gfCNCPoint6[7271] = {X 240.3232, Y 30.5783, Z -8.0000, A 0.000, B 0.000, C 0.000 }
gfCNCPoint6[7272] = {X 239.3655, Y 29.5329, Z -8.0000, A 0.000, B 0.000, C 0.000 }
gfCNCPoint6[7273] = {X 238.5491, Y 28.3738, Z -8.0000, A 0.000, B 0.000, C 0.000 }
gfCNCPoint6[7274] = {X 237.8873, Y 27.1200, Z -8.0000, A 0.000, B 0.000, C 0.000 }
gfCNCPoint6[7275] = {X 237.3910, Y 25.7920, Z -8.0000, A 0.000, B 0.000, C 0.000 }
gfCNCPoint6[7276] = {X 236.9772, Y 24.0072, Z -8.0000, A 0.000, B 0.000, C 0.000 }
gfCNCPoint6[7277] = {X 236.7665, Y 22.1872, Z -8.0000, A 0.000, B 0.000, C 0.000 }
gfCNCPoint6[7278] = {X 236.7613, Y 20.3551, Z -8.0000, A 0.000, B 0.000, C 0.000 }
gfCNCPoint6[7279] = {X 236.9619, Y 18.5340, Z -8.0000, A 0.000, B 0.000, C 0.000 }
gfCNCPoint6[7280] = {X 237.3656, Y 16.7468, Z -8.0000, A 0.000, B 0.000, C 0.000 }
gfCNCPoint6[7281] = {X 237.9247, Y 15.2027, Z -8.0000, A 0.000, B 0.000, C 0.000 }
gfCNCPoint6[7282] = {X 238.6960, Y 13.7528, Z -8.0000, A 0.000, B 0.000, C 0.000 }
gfCNCPoint6[7283] = {X 239.6641, Y 12.4263, Z -8.0000, A 0.000, B 0.000, C 0.000 }
gfCNCPoint6[7284] = {X 240.8097, Y 11.2496, Z -8.0000, A 0.000, B 0.000, C 0.000 }
gfCNCPoint6[7285] = {X 242.1099, Y 10.2463, Z -8.0000, A 0.000, B 0.000, C 0.000 }
gfCNCPoint6[7286] = {X 243.5386, Y 9.4365, Z -8.0000, A 0.000, B 0.000, C 0.000 }
gfCNCPoint6[7287] = {X 245.0673, Y 8.8364, Z -8.0000, A 0.000, B 0.000, C 0.000 }
gfCNCPoint6[7288] = {X 246.6653, Y 8.4579, Z -8.0000, A 0.000, B 0.000, C 0.000 }
gfCNCPoint6[7289] = {X 248.7417, Y 8.1890, Z -8.0000, A 0.000, B 0.000, C 0.000 }
gfCNCPoint6[7290] = {X 250.8340, Y 8.1092, Z -8.0000, A 0.000, B 0.000, C 0.000 }
gfCNCPoint6[7291] = {X 266.7614, Y 8.1092, Z -8.0000, A 0.000, B 0.000, C 0.000 }
gfCNCPoint6[7292] = {X 267.6638, Y 8.2176, Z -8.0000, A 0.000, B 0.000, C 0.000 }
gfCNCPoint6[7293] = {X 268.5198, Y 8.5230, Z -8.0000, A 0.000, B 0.000, C 0.000 }
gfCNCPoint6[7294] = {X 269.2870, Y 9.0102, Z -8.0000, A 0.000, B 0.000, C 0.000 }
gfCNCPoint6[7295] = {X 269.9275, Y 9.6550, Z -8.0000, A 0.000, B 0.000, C 0.000 }
gfCNCPoint6[7296] = {X 270.4094, Y 10.4256, Z -8.0000, A 0.000, B 0.000, C 0.000 }
gfCNCPoint6[7297] = {X 270.7088, Y 11.2837, Z -8.0000, A 0.000, B 0.000, C 0.000 }
gfCNCPoint6[7298] = {X 270.8110, Y 12.1867, Z -8.0000, A 0.000, B 0.000, C 0.000 }
gfCNCPoint6[7299] = {X 270.8108, Y 13.0200, Z -8.0000, A 0.000, B 0.000, C 0.000 }
gfCNCPoint6[7300] = {X 270.7023, Y 13.9135, Z -8.0000, A 0.000, B 0.000, C 0.000 }
gfCNCPoint6[7301] = {X 270.4006, Y 14.7615, Z -8.0000, A 0.000, B 0.000, C 0.000 }
gfCNCPoint6[7302] = {X 269.9202, Y 15.5227, Z -8.0000, A 0.000, B 0.000, C 0.000 }
gfCNCPoint6[7303] = {X 269.2847, Y 16.1601, Z -8.0000, A 0.000, B 0.000, C 0.000 }
gfCNCPoint6[7304] = {X 269.2849, Y 28.5938, Z -8.0000, A 0.000, B 0.000, C 0.000 }
gfCNCPoint6[7305] = {X 273.2849, Y 28.5937, Z -8.0000, A 0.000, B 0.000, C 0.000 }
gfCNCPoint6[7306] = {X 269.2049, Y 28.5938, Z -8.0000, A 0.000, B 0.000, C 0.000 }
gfCNCPoint6[7307] = {X 269.2051, Y 41.0652, Z -8.0000, A 0.000, B 0.000, C 0.000 }
gfCNCPoint6[7308] = {X 269.3438, Y 41.1800, Z -8.0000, A 0.000, B 0.000, C 0.000 }
gfCNCPoint6[7309] = {X 269.9292, Y 41.8064, Z -8.0000, A 0.000, B 0.000, C 0.000 }
gfCNCPoint6[7310] = {X 270.3677, Y 42.5431, Z -8.0000, A 0.000, B 0.000, C 0.000 }
gfCNCPoint6[7311] = {X 270.6392, Y 43.3564, Z -8.0000, A 0.000, B 0.000, C 0.000 }
gfCNCPoint6[7312] = {X 270.7310, Y 44.2089, Z -8.0000, A 0.000, B 0.000, C 0.000 }
gfCNCPoint6[7313] = {X 270.7310, Y 45.0000, Z -8.0000, A 0.000, B 0.000, C 0.000 }
gfCNCPoint6[7314] = {X 270.6307, Y 45.8901, Z -8.0000, A 0.000, B 0.000, C 0.000 }
gfCNCPoint6[7315] = {X 270.3349, Y 46.7355, Z -8.0000, A 0.000, B 0.000, C 0.000 }
gfCNCPoint6[7316] = {X 269.8584, Y 47.4940, Z -8.0000, A 0.000, B 0.000, C 0.000 }
gfCNCPoint6[7317] = {X 269.2250, Y 48.1273, Z -8.0000, A 0.000, B 0.000, C 0.000 }
gfCNCPoint6[7318] = {X 268.4666, Y 48.6039, Z -8.0000, A 0.000, B 0.000, C 0.000 }
gfCNCPoint6[7319] = {X 267.6211, Y 48.8997, Z -8.0000, A 0.000, B 0.000, C 0.000 }
gfCNCPoint6[7320] = {X 266.7310, Y 49.0000, Z -8.0000, A 0.000, B 0.000, C 0.000 }
gfCNCPoint6[7321] = {X 260.2876, Y 49.0000, Z -8.0000, A 0.000, B 0.000, C 0.000 }
gfCNCPoint6[7322] = {X 259.3975, Y 48.8997, Z -8.0000, A 0.000, B 0.000, C 0.000 }
gfCNCPoint6[7323] = {X 258.5520, Y 48.6039, Z -8.0000, A 0.000, B 0.000, C 0.000 }
gfCNCPoint6[7324] = {X 257.7936, Y 48.1273, Z -8.0000, A 0.000, B 0.000, C 0.000 }
gfCNCPoint6[7325] = {X 257.1602, Y 47.4939, Z -8.0000, A 0.000, B 0.000, C 0.000 }
gfCNCPoint6[7326] = {X 256.6837, Y 46.7355, Z -8.0000, A 0.000, B 0.000, C 0.000 }
gfCNCPoint6[7327] = {X 256.3878, Y 45.8901, Z -8.0000, A 0.000, B 0.000, C 0.000 }
gfCNCPoint6[7328] = {X 256.2876, Y 45.0000, Z -8.0000, A 0.000, B 0.000, C 0.000 }
gfCNCPoint6[7329] = {X 256.2879, Y 44.1538, Z -8.0000, A 0.000, B 0.000, C 0.000 }
gfCNCPoint6[7330] = {X 256.3986, Y 43.2730, Z -8.0000, A 0.000, B 0.000, C 0.000 }
gfCNCPoint6[7331] = {X 256.7008, Y 42.4382, Z -8.0000, A 0.000, B 0.000, C 0.000 }
gfCNCPoint6[7332] = {X 257.1796, Y 41.6907, Z -8.0000, A 0.000, B 0.000, C 0.000 }
gfCNCPoint6[7333] = {X 257.8115, Y 41.0672, Z -8.0000, A 0.000, B 0.000, C 0.000 }
gfCNCPoint6[7334] = {X 257.8115, Y 34.1538, Z -8.0000, A 0.000, B 0.000, C 0.000 }
gfCNCPoint6[7335] = {X 254.8178, Y 34.1538, Z -8.0000, A 0.000, B 0.000, C 0.000 }
gfCNCPoint6[7336] = {X 254.5738, Y 34.1534, Z -8.0000, A 0.000, B 0.000, C 0.000 }
gfCNCPoint6[7337] = {X 250.1360, Y 42.7967, Z -8.0000, A 0.000, B 0.000, C 0.000 }
gfCNCPoint6[7338] = {X 250.3287, Y 43.4911, Z -8.0000, A 0.000, B 0.000, C 0.000 }
gfCNCPoint6[7339] = {X 250.3936, Y 44.2089, Z -8.0000, A 0.000, B 0.000, C 0.000 }
gfCNCPoint6[7340] = {X 250.3936, Y 45.0000, Z -8.0000, A 0.000, B 0.000, C 0.000 }
gfCNCPoint6[7341] = {X 250.2933, Y 45.8901, Z -8.0000, A 0.000, B 0.000, C 0.000 }
gfCNCPoint6[7342] = {X 249.9974, Y 46.7355, Z -8.0000, A 0.000, B 0.000, C 0.000 }
gfCNCPoint6[7343] = {X 249.5209, Y 47.4940, Z -8.0000, A 0.000, B 0.000, C 0.000 }
gfCNCPoint6[7344] = {X 248.8875, Y 48.1273, Z -8.0000, A 0.000, B 0.000, C 0.000 }
gfCNCPoint6[7345] = {X 248.1291, Y 48.6039, Z -8.0000, A 0.000, B 0.000, C 0.000 }
gfCNCPoint6[7346] = {X 247.2836, Y 48.8997, Z -8.0000, A 0.000, B 0.000, C 0.000 }
gfCNCPoint6[7347] = {X 246.3936, Y 49.0000, Z -8.0000, A 0.000, B 0.000, C 0.000 }
gfCNCPoint6[7348] = {X 239.8075, Y 49.0000, Z -8.0000, A 0.000, B 0.000, C 0.000 }
gfCNCPoint6[7349] = {X 238.9174, Y 48.8997, Z -8.0000, A 0.000, B 0.000, C 0.000 }
gfCNCPoint6[7350] = {X 238.0720, Y 48.6039, Z -8.0000, A 0.000, B 0.000, C 0.000 }
gfCNCPoint6[7351] = {X 237.3135, Y 48.1273, Z -8.0000, A 0.000, B 0.000, C 0.000 }
gfCNCPoint6[7352] = {X 236.6802, Y 47.4940, Z -8.0000, A 0.000, B 0.000, C 0.000 }
gfCNCPoint6[7353] = {X 236.2036, Y 46.7355, Z -8.0000, A 0.000, B 0.000, C 0.000 }
gfCNCPoint6[7354] = {X 235.9078, Y 45.8901, Z -8.0000, A 0.000, B 0.000, C 0.000 }
gfCNCPoint6[7355] = {X 235.8075, Y 45.0000, Z -8.0000, A 0.000, B 0.000, C 0.000 }
gfCNCPoint6[7356] = {X 235.8079, Y 44.1538, Z -8.0000, A 0.000, B 0.000, C 0.000 }
gfCNCPoint6[7357] = {X 235.9027, Y 43.3414, Z -8.0000, A 0.000, B 0.000, C 0.000 }
gfCNCPoint6[7358] = {X 236.1607, Y 42.5654, Z -8.0000, A 0.000, B 0.000, C 0.000 }
gfCNCPoint6[7359] = {X 236.5712, Y 41.8580, Z -8.0000, A 0.000, B 0.000, C 0.000 }
gfCNCPoint6[7360] = {X 237.1169, Y 41.2489, Z -8.0000, A 0.000, B 0.000, C 0.000 }
gfCNCPoint6[7361] = {X 237.7752, Y 40.7635, Z -8.0000, A 0.000, B 0.000, C 0.000 }
gfCNCPoint6[7362] = {X 238.5184, Y 40.4222, Z -8.0000, A 0.000, B 0.000, C 0.000 }
gfCNCPoint6[7363] = {X 242.7041, Y 32.2292, Z -8.0000, A 0.000, B 0.000, C 0.000 }
gfCNCPoint6[7364] = {X 241.5058, Y 31.4666, Z -8.0000, A 0.000, B 0.000, C 0.000 }
gfCNCPoint6[7365] = {X 240.4158, Y 30.5561, Z -8.0000, A 0.000, B 0.000, C 0.000 }
gfCNCPoint6[7366] = {X 239.4521, Y 29.5127, Z -8.0000, A 0.000, B 0.000, C 0.000 }
gfCNCPoint6[7367] = {X 238.6308, Y 28.3539, Z -8.0000, A 0.000, B 0.000, C 0.000 }
gfCNCPoint6[7368] = {X 237.9656, Y 27.0990, Z -8.0000, A 0.000, B 0.000, C 0.000 }
gfCNCPoint6[7369] = {X 237.4676, Y 25.7689, Z -8.0000, A 0.000, B 0.000, C 0.000 }
gfCNCPoint6[7370] = {X 237.0560, Y 23.9929, Z -8.0000, A 0.000, B 0.000, C 0.000 }
gfCNCPoint6[7371] = {X 236.8463, Y 22.1820, Z -8.0000, A 0.000, B 0.000, C 0.000 }
gfCNCPoint6[7372] = {X 236.8412, Y 20.3590, Z -8.0000, A 0.000, B 0.000, C 0.000 }
gfCNCPoint6[7373] = {X 237.0408, Y 18.5469, Z -8.0000, A 0.000, B 0.000, C 0.000 }
gfCNCPoint6[7374] = {X 237.4426, Y 16.7687, Z -8.0000, A 0.000, B 0.000, C 0.000 }
gfCNCPoint6[7375] = {X 237.9978, Y 15.2351, Z -8.0000, A 0.000, B 0.000, C 0.000 }
gfCNCPoint6[7376] = {X 238.7638, Y 13.7952, Z -8.0000, A 0.000, B 0.000, C 0.000 }
gfCNCPoint6[7377] = {X 239.7254, Y 12.4778, Z -8.0000, A 0.000, B 0.000, C 0.000 }
gfCNCPoint6[7378] = {X 240.8631, Y 11.3092, Z -8.0000, A 0.000, B 0.000, C 0.000 }
gfCNCPoint6[7379] = {X 242.1544, Y 10.3128, Z -8.0000, A 0.000, B 0.000, C 0.000 }
gfCNCPoint6[7380] = {X 243.5734, Y 9.5086, Z -8.0000, A 0.000, B 0.000, C 0.000 }
gfCNCPoint6[7381] = {X 245.0916, Y 8.9126, Z -8.0000, A 0.000, B 0.000, C 0.000 }
gfCNCPoint6[7382] = {X 246.6787, Y 8.5367, Z -8.0000, A 0.000, B 0.000, C 0.000 }
gfCNCPoint6[7383] = {X 248.7483, Y 8.2687, Z -8.0000, A 0.000, B 0.000, C 0.000 }
gfCNCPoint6[7384] = {X 250.8336, Y 8.1892, Z -8.0000, A 0.000, B 0.000, C 0.000 }
gfCNCPoint6[7385] = {X 266.7608, Y 8.1892, Z -8.0000, A 0.000, B 0.000, C 0.000 }
gfCNCPoint6[7386] = {X 267.6454, Y 8.2955, Z -8.0000, A 0.000, B 0.000, C 0.000 }
gfCNCPoint6[7387] = {X 268.4847, Y 8.5949, Z -8.0000, A 0.000, B 0.000, C 0.000 }
gfCNCPoint6[7388] = {X 269.2369, Y 9.0725, Z -8.0000, A 0.000, B 0.000, C 0.000 }
gfCNCPoint6[7389] = {X 269.8648, Y 9.7047, Z -8.0000, A 0.000, B 0.000, C 0.000 }
gfCNCPoint6[7390] = {X 270.3372, Y 10.4602, Z -8.0000, A 0.000, B 0.000, C 0.000 }
gfCNCPoint6[7391] = {X 270.6308, Y 11.3015, Z -8.0000, A 0.000, B 0.000, C 0.000 }
gfCNCPoint6[7392] = {X 270.7310, Y 12.1868, Z -8.0000, A 0.000, B 0.000, C 0.000 }
gfCNCPoint6[7393] = {X 270.7308, Y 13.0192, Z -8.0000, A 0.000, B 0.000, C 0.000 }
gfCNCPoint6[7394] = {X 270.6223, Y 13.9045, Z -8.0000, A 0.000, B 0.000, C 0.000 }
gfCNCPoint6[7395] = {X 270.3202, Y 14.7437, Z -8.0000, A 0.000, B 0.000, C 0.000 }
gfCNCPoint6[7396] = {X 269.8397, Y 15.4952, Z -8.0000, A 0.000, B 0.000, C 0.000 }
gfCNCPoint6[7397] = {X 269.2047, Y 16.1215, Z -8.0000, A 0.000, B 0.000, C 0.000 }
gfCNCPoint6[7398] = {X 269.2049, Y 28.5938, Z -8.0000, A 0.000, B 0.000, C 0.000 }
gfCNCPoint6[7399] = {X 273.2849, Y 28.5937, Z -8.0000, A 0.000, B 0.000, C 0.000 }
gfCNCPoint6[7400] = {X 273.2849, Y 28.5937, Z -5.0000, A 0.000, B 0.000, C 0.000 }
gfCNCPoint6[7401] = {X 273.2849, Y 28.5937, Z 11.0000, A 0.000, B 0.000, C 0.000 }
gfCNCPoint6[7402] = {X 277.7442, Y 28.5918, Z 11.0000, A 0.000, B 0.000, C 0.000 }
gfCNCPoint6[7403] = {X 277.7442, Y 28.5918, Z -5.0000, A 0.000, B 0.000, C 0.000 }
gfCNCPoint6[7404] = {X 277.7442, Y 28.5918, Z -8.0000, A 0.000, B 0.000, C 0.000 }
gfCNCPoint6[7405] = {X 281.8242, Y 28.5918, Z -8.0000, A 0.000, B 0.000, C 0.000 }
gfCNCPoint6[7406] = {X 281.8243, Y 16.2734, Z -8.0000, A 0.000, B 0.000, C 0.000 }
gfCNCPoint6[7407] = {X 281.1862, Y 15.6023, Z -8.0000, A 0.000, B 0.000, C 0.000 }
gfCNCPoint6[7408] = {X 280.7057, Y 14.8107, Z -8.0000, A 0.000, B 0.000, C 0.000 }
gfCNCPoint6[7409] = {X 280.4050, Y 13.9349, Z -8.0000, A 0.000, B 0.000, C 0.000 }
gfCNCPoint6[7410] = {X 280.2978, Y 13.0151, Z -8.0000, A 0.000, B 0.000, C 0.000 }
gfCNCPoint6[7411] = {X 280.2977, Y 12.1868, Z -8.0000, A 0.000, B 0.000, C 0.000 }
gfCNCPoint6[7412] = {X 280.4060, Y 11.2255, Z -8.0000, A 0.000, B 0.000, C 0.000 }
gfCNCPoint6[7413] = {X 280.7255, Y 10.3124, Z -8.0000, A 0.000, B 0.000, C 0.000 }
gfCNCPoint6[7414] = {X 281.2402, Y 9.4933, Z -8.0000, A 0.000, B 0.000, C 0.000 }
gfCNCPoint6[7415] = {X 281.9242, Y 8.8093, Z -8.0000, A 0.000, B 0.000, C 0.000 }
gfCNCPoint6[7416] = {X 282.7433, Y 8.2946, Z -8.0000, A 0.000, B 0.000, C 0.000 }
gfCNCPoint6[7417] = {X 283.6564, Y 7.9751, Z -8.0000, A 0.000, B 0.000, C 0.000 }
gfCNCPoint6[7418] = {X 284.6177, Y 7.8668, Z -8.0000, A 0.000, B 0.000, C 0.000 }
gfCNCPoint6[7419] = {X 291.0611, Y 7.8668, Z -8.0000, A 0.000, B 0.000, C 0.000 }
gfCNCPoint6[7420] = {X 292.0224, Y 7.9751, Z -8.0000, A 0.000, B 0.000, C 0.000 }
gfCNCPoint6[7421] = {X 292.9355, Y 8.2946, Z -8.0000, A 0.000, B 0.000, C 0.000 }
gfCNCPoint6[7422] = {X 293.7546, Y 8.8093, Z -8.0000, A 0.000, B 0.000, C 0.000 }
gfCNCPoint6[7423] = {X 294.4386, Y 9.4933, Z -8.0000, A 0.000, B 0.000, C 0.000 }
gfCNCPoint6[7424] = {X 294.9533, Y 10.3124, Z -8.0000, A 0.000, B 0.000, C 0.000 }
gfCNCPoint6[7425] = {X 295.2728, Y 11.2255, Z -8.0000, A 0.000, B 0.000, C 0.000 }
gfCNCPoint6[7426] = {X 295.3811, Y 12.1868, Z -8.0000, A 0.000, B 0.000, C 0.000 }
gfCNCPoint6[7427] = {X 295.3811, Y 12.9782, Z -8.0000, A 0.000, B 0.000, C 0.000 }
gfCNCPoint6[7428] = {X 295.2798, Y 13.9077, Z -8.0000, A 0.000, B 0.000, C 0.000 }
gfCNCPoint6[7429] = {X 294.9809, Y 14.7936, Z -8.0000, A 0.000, B 0.000, C 0.000 }
gfCNCPoint6[7430] = {X 294.4983, Y 15.5945, Z -8.0000, A 0.000, B 0.000, C 0.000 }
gfCNCPoint6[7431] = {X 293.8548, Y 16.2728, Z -8.0000, A 0.000, B 0.000, C 0.000 }
gfCNCPoint6[7432] = {X 293.8557, Y 22.1965, Z -8.0000, A 0.000, B 0.000, C 0.000 }
gfCNCPoint6[7433] = {X 302.7582, Y 22.1965, Z -8.0000, A 0.000, B 0.000, C 0.000 }
gfCNCPoint6[7434] = {X 302.7633, Y 16.2771, Z -8.0000, A 0.000, B 0.000, C 0.000 }
gfCNCPoint6[7435] = {X 302.1236, Y 15.6061, Z -8.0000, A 0.000, B 0.000, C 0.000 }
gfCNCPoint6[7436] = {X 301.6418, Y 14.8140, Z -8.0000, A 0.000, B 0.000, C 0.000 }
gfCNCPoint6[7437] = {X 301.3401, Y 13.9374, Z -8.0000, A 0.000, B 0.000, C 0.000 }
gfCNCPoint6[7438] = {X 301.2324, Y 13.0165, Z -8.0000, A 0.000, B 0.000, C 0.000 }
gfCNCPoint6[7439] = {X 301.2323, Y 12.1868, Z -8.0000, A 0.000, B 0.000, C 0.000 }
gfCNCPoint6[7440] = {X 301.3406, Y 11.2255, Z -8.0000, A 0.000, B 0.000, C 0.000 }
gfCNCPoint6[7441] = {X 301.6601, Y 10.3124, Z -8.0000, A 0.000, B 0.000, C 0.000 }
gfCNCPoint6[7442] = {X 302.1747, Y 9.4933, Z -8.0000, A 0.000, B 0.000, C 0.000 }
gfCNCPoint6[7443] = {X 302.8588, Y 8.8093, Z -8.0000, A 0.000, B 0.000, C 0.000 }
gfCNCPoint6[7444] = {X 303.6779, Y 8.2946, Z -8.0000, A 0.000, B 0.000, C 0.000 }
gfCNCPoint6[7445] = {X 304.5910, Y 7.9751, Z -8.0000, A 0.000, B 0.000, C 0.000 }
gfCNCPoint6[7446] = {X 305.5523, Y 7.8668, Z -8.0000, A 0.000, B 0.000, C 0.000 }
gfCNCPoint6[7447] = {X 311.9957, Y 7.8668, Z -8.0000, A 0.000, B 0.000, C 0.000 }
gfCNCPoint6[7448] = {X 312.9570, Y 7.9751, Z -8.0000, A 0.000, B 0.000, C 0.000 }
gfCNCPoint6[7449] = {X 313.8701, Y 8.2946, Z -8.0000, A 0.000, B 0.000, C 0.000 }
gfCNCPoint6[7450] = {X 314.6892, Y 8.8093, Z -8.0000, A 0.000, B 0.000, C 0.000 }
gfCNCPoint6[7451] = {X 315.3732, Y 9.4933, Z -8.0000, A 0.000, B 0.000, C 0.000 }
gfCNCPoint6[7452] = {X 315.8879, Y 10.3124, Z -8.0000, A 0.000, B 0.000, C 0.000 }
gfCNCPoint6[7453] = {X 316.2074, Y 11.2255, Z -8.0000, A 0.000, B 0.000, C 0.000 }
gfCNCPoint6[7454] = {X 316.3157, Y 12.1868, Z -8.0000, A 0.000, B 0.000, C 0.000 }
gfCNCPoint6[7455] = {X 316.3157, Y 12.9782, Z -8.0000, A 0.000, B 0.000, C 0.000 }
gfCNCPoint6[7456] = {X 316.2145, Y 13.9077, Z -8.0000, A 0.000, B 0.000, C 0.000 }
gfCNCPoint6[7457] = {X 315.9156, Y 14.7937, Z -8.0000, A 0.000, B 0.000, C 0.000 }
gfCNCPoint6[7458] = {X 315.4331, Y 15.5947, Z -8.0000, A 0.000, B 0.000, C 0.000 }
gfCNCPoint6[7459] = {X 314.7895, Y 16.2730, Z -8.0000, A 0.000, B 0.000, C 0.000 }
gfCNCPoint6[7460] = {X 314.7893, Y 40.9136, Z -8.0000, A 0.000, B 0.000, C 0.000 }
gfCNCPoint6[7461] = {X 315.4273, Y 41.5845, Z -8.0000, A 0.000, B 0.000, C 0.000 }
gfCNCPoint6[7462] = {X 315.9077, Y 42.3760, Z -8.0000, A 0.000, B 0.000, C 0.000 }
gfCNCPoint6[7463] = {X 316.2084, Y 43.2517, Z -8.0000, A 0.000, B 0.000, C 0.000 }
gfCNCPoint6[7464] = {X 316.3156, Y 44.1713, Z -8.0000, A 0.000, B 0.000, C 0.000 }
gfCNCPoint6[7465] = {X 316.3157, Y 45.0000, Z -8.0000, A 0.000, B 0.000, C 0.000 }
gfCNCPoint6[7466] = {X 316.2074, Y 45.9613, Z -8.0000, A 0.000, B 0.000, C 0.000 }
gfCNCPoint6[7467] = {X 315.8879, Y 46.8744, Z -8.0000, A 0.000, B 0.000, C 0.000 }
gfCNCPoint6[7468] = {X 315.3732, Y 47.6935, Z -8.0000, A 0.000, B 0.000, C 0.000 }
gfCNCPoint6[7469] = {X 314.6892, Y 48.3775, Z -8.0000, A 0.000, B 0.000, C 0.000 }
gfCNCPoint6[7470] = {X 313.8701, Y 48.8922, Z -8.0000, A 0.000, B 0.000, C 0.000 }
gfCNCPoint6[7471] = {X 312.9570, Y 49.2117, Z -8.0000, A 0.000, B 0.000, C 0.000 }
gfCNCPoint6[7472] = {X 311.9957, Y 49.3200, Z -8.0000, A 0.000, B 0.000, C 0.000 }
gfCNCPoint6[7473] = {X 305.5523, Y 49.3200, Z -8.0000, A 0.000, B 0.000, C 0.000 }
gfCNCPoint6[7474] = {X 304.5958, Y 49.2128, Z -8.0000, A 0.000, B 0.000, C 0.000 }
gfCNCPoint6[7475] = {X 303.6868, Y 48.8965, Z -8.0000, A 0.000, B 0.000, C 0.000 }
gfCNCPoint6[7476] = {X 302.8704, Y 48.3868, Z -8.0000, A 0.000, B 0.000, C 0.000 }
gfCNCPoint6[7477] = {X 302.1872, Y 47.7090, Z -8.0000, A 0.000, B 0.000, C 0.000 }
gfCNCPoint6[7478] = {X 301.6709, Y 46.8967, Z -8.0000, A 0.000, B 0.000, C 0.000 }
gfCNCPoint6[7479] = {X 301.3473, Y 45.9903, Z -8.0000, A 0.000, B 0.000, C 0.000 }
gfCNCPoint6[7480] = {X 301.2324, Y 45.0348, Z -8.0000, A 0.000, B 0.000, C 0.000 }
gfCNCPoint6[7481] = {X 301.2323, Y 44.2015, Z -8.0000, A 0.000, B 0.000, C 0.000 }
gfCNCPoint6[7482] = {X 301.3493, Y 43.2653, Z -8.0000, A 0.000, B 0.000, C 0.000 }
gfCNCPoint6[7483] = {X 301.6520, Y 42.3718, Z -8.0000, A 0.000, B 0.000, C 0.000 }
gfCNCPoint6[7484] = {X 302.1282, Y 41.5574, Z -8.0000, A 0.000, B 0.000, C 0.000 }
gfCNCPoint6[7485] = {X 302.7584, Y 40.8553, Z -8.0000, A 0.000, B 0.000, C 0.000 }
gfCNCPoint6[7486] = {X 302.7584, Y 34.0343, Z -8.0000, A 0.000, B 0.000, C 0.000 }
gfCNCPoint6[7487] = {X 293.8554, Y 34.0343, Z -8.0000, A 0.000, B 0.000, C 0.000 }
gfCNCPoint6[7488] = {X 293.8549, Y 40.9018, Z -8.0000, A 0.000, B 0.000, C 0.000 }
gfCNCPoint6[7489] = {X 294.4941, Y 41.5858, Z -8.0000, A 0.000, B 0.000, C 0.000 }
gfCNCPoint6[7490] = {X 294.9746, Y 42.3894, Z -8.0000, A 0.000, B 0.000, C 0.000 }
gfCNCPoint6[7491] = {X 295.2748, Y 43.2762, Z -8.0000, A 0.000, B 0.000, C 0.000 }
gfCNCPoint6[7492] = {X 295.3811, Y 44.2064, Z -8.0000, A 0.000, B 0.000, C 0.000 }
gfCNCPoint6[7493] = {X 295.3811, Y 45.0000, Z -8.0000, A 0.000, B 0.000, C 0.000 }
gfCNCPoint6[7494] = {X 295.2728, Y 45.9613, Z -8.0000, A 0.000, B 0.000, C 0.000 }
gfCNCPoint6[7495] = {X 294.9533, Y 46.8744, Z -8.0000, A 0.000, B 0.000, C 0.000 }
gfCNCPoint6[7496] = {X 294.4386, Y 47.6935, Z -8.0000, A 0.000, B 0.000, C 0.000 }
gfCNCPoint6[7497] = {X 293.7546, Y 48.3775, Z -8.0000, A 0.000, B 0.000, C 0.000 }
gfCNCPoint6[7498] = {X 292.9355, Y 48.8922, Z -8.0000, A 0.000, B 0.000, C 0.000 }
gfCNCPoint6[7499] = {X 292.0224, Y 49.2117, Z -8.0000, A 0.000, B 0.000, C 0.000 }
gfCNCPoint6[7500] = {X 291.0611, Y 49.3200, Z -8.0000, A 0.000, B 0.000, C 0.000 }
gfCNCPoint6[7501] = {X 284.6177, Y 49.3200, Z -8.0000, A 0.000, B 0.000, C 0.000 }
gfCNCPoint6[7502] = {X 283.6613, Y 49.2128, Z -8.0000, A 0.000, B 0.000, C 0.000 }
gfCNCPoint6[7503] = {X 282.7524, Y 48.8965, Z -8.0000, A 0.000, B 0.000, C 0.000 }
gfCNCPoint6[7504] = {X 281.9360, Y 48.3869, Z -8.0000, A 0.000, B 0.000, C 0.000 }
gfCNCPoint6[7505] = {X 281.2527, Y 47.7092, Z -8.0000, A 0.000, B 0.000, C 0.000 }
gfCNCPoint6[7506] = {X 280.7365, Y 46.8970, Z -8.0000, A 0.000, B 0.000, C 0.000 }
gfCNCPoint6[7507] = {X 280.4128, Y 45.9907, Z -8.0000, A 0.000, B 0.000, C 0.000 }
gfCNCPoint6[7508] = {X 280.2978, Y 45.0352, Z -8.0000, A 0.000, B 0.000, C 0.000 }
gfCNCPoint6[7509] = {X 280.2977, Y 44.2075, Z -8.0000, A 0.000, B 0.000, C 0.000 }
gfCNCPoint6[7510] = {X 280.4017, Y 43.2782, Z -8.0000, A 0.000, B 0.000, C 0.000 }
gfCNCPoint6[7511] = {X 280.7014, Y 42.3925, Z -8.0000, A 0.000, B 0.000, C 0.000 }
gfCNCPoint6[7512] = {X 281.1829, Y 41.5909, Z -8.0000, A 0.000, B 0.000, C 0.000 }
gfCNCPoint6[7513] = {X 281.8241, Y 40.9103, Z -8.0000, A 0.000, B 0.000, C 0.000 }
gfCNCPoint6[7514] = {X 281.8242, Y 28.5918, Z -8.0000, A 0.000, B 0.000, C 0.000 }
gfCNCPoint6[7515] = {X 277.8242, Y 28.5918, Z -8.0000, A 0.000, B 0.000, C 0.000 }
gfCNCPoint6[7516] = {X 281.9042, Y 28.5918, Z -8.0000, A 0.000, B 0.000, C 0.000 }
gfCNCPoint6[7517] = {X 281.9043, Y 16.2361, Z -8.0000, A 0.000, B 0.000, C 0.000 }
gfCNCPoint6[7518] = {X 281.2666, Y 15.5757, Z -8.0000, A 0.000, B 0.000, C 0.000 }
gfCNCPoint6[7519] = {X 280.7860, Y 14.7935, Z -8.0000, A 0.000, B 0.000, C 0.000 }
gfCNCPoint6[7520] = {X 280.4850, Y 13.9262, Z -8.0000, A 0.000, B 0.000, C 0.000 }
gfCNCPoint6[7521] = {X 280.3778, Y 13.0144, Z -8.0000, A 0.000, B 0.000, C 0.000 }
gfCNCPoint6[7522] = {X 280.3777, Y 12.1868, Z -8.0000, A 0.000, B 0.000, C 0.000 }
gfCNCPoint6[7523] = {X 280.4840, Y 11.2433, Z -8.0000, A 0.000, B 0.000, C 0.000 }
gfCNCPoint6[7524] = {X 280.7976, Y 10.3472, Z -8.0000, A 0.000, B 0.000, C 0.000 }
gfCNCPoint6[7525] = {X 281.3027, Y 9.5432, Z -8.0000, A 0.000, B 0.000, C 0.000 }
gfCNCPoint6[7526] = {X 281.9741, Y 8.8719, Z -8.0000, A 0.000, B 0.000, C 0.000 }
gfCNCPoint6[7527] = {X 282.7780, Y 8.3667, Z -8.0000, A 0.000, B 0.000, C 0.000 }
gfCNCPoint6[7528] = {X 283.6742, Y 8.0531, Z -8.0000, A 0.000, B 0.000, C 0.000 }
gfCNCPoint6[7529] = {X 284.6177, Y 7.9468, Z -8.0000, A 0.000, B 0.000, C 0.000 }
gfCNCPoint6[7530] = {X 291.0611, Y 7.9468, Z -8.0000, A 0.000, B 0.000, C 0.000 }
gfCNCPoint6[7531] = {X 292.0046, Y 8.0531, Z -8.0000, A 0.000, B 0.000, C 0.000 }
gfCNCPoint6[7532] = {X 292.9008, Y 8.3667, Z -8.0000, A 0.000, B 0.000, C 0.000 }
gfCNCPoint6[7533] = {X 293.7047, Y 8.8718, Z -8.0000, A 0.000, B 0.000, C 0.000 }
gfCNCPoint6[7534] = {X 294.3761, Y 9.5432, Z -8.0000, A 0.000, B 0.000, C 0.000 }
gfCNCPoint6[7535] = {X 294.8812, Y 10.3471, Z -8.0000, A 0.000, B 0.000, C 0.000 }
gfCNCPoint6[7536] = {X 295.1948, Y 11.2433, Z -8.0000, A 0.000, B 0.000, C 0.000 }
gfCNCPoint6[7537] = {X 295.3011, Y 12.1868, Z -8.0000, A 0.000, B 0.000, C 0.000 }
gfCNCPoint6[7538] = {X 295.3011, Y 12.9782, Z -8.0000, A 0.000, B 0.000, C 0.000 }
gfCNCPoint6[7539] = {X 295.1997, Y 13.8995, Z -8.0000, A 0.000, B 0.000, C 0.000 }
gfCNCPoint6[7540] = {X 294.9005, Y 14.7767, Z -8.0000, A 0.000, B 0.000, C 0.000 }
gfCNCPoint6[7541] = {X 294.4178, Y 15.5680, Z -8.0000, A 0.000, B 0.000, C 0.000 }
gfCNCPoint6[7542] = {X 293.7748, Y 16.2355, Z -8.0000, A 0.000, B 0.000, C 0.000 }
gfCNCPoint6[7543] = {X 293.7757, Y 22.2765, Z -8.0000, A 0.000, B 0.000, C 0.000 }
gfCNCPoint6[7544] = {X 302.8381, Y 22.2765, Z -8.0000, A 0.000, B 0.000, C 0.000 }
gfCNCPoint6[7545] = {X 302.8433, Y 16.2398, Z -8.0000, A 0.000, B 0.000, C 0.000 }
gfCNCPoint6[7546] = {X 302.2041, Y 15.5794, Z -8.0000, A 0.000, B 0.000, C 0.000 }
gfCNCPoint6[7547] = {X 301.7221, Y 14.7968, Z -8.0000, A 0.000, B 0.000, C 0.000 }
gfCNCPoint6[7548] = {X 301.4202, Y 13.9286, Z -8.0000, A 0.000, B 0.000, C 0.000 }
gfCNCPoint6[7549] = {X 301.3124, Y 13.0158, Z -8.0000, A 0.000, B 0.000, C 0.000 }
gfCNCPoint6[7550] = {X 301.3123, Y 12.1868, Z -8.0000, A 0.000, B 0.000, C 0.000 }
gfCNCPoint6[7551] = {X 301.4186, Y 11.2433, Z -8.0000, A 0.000, B 0.000, C 0.000 }
gfCNCPoint6[7552] = {X 301.7321, Y 10.3471, Z -8.0000, A 0.000, B 0.000, C 0.000 }
gfCNCPoint6[7553] = {X 302.2373, Y 9.5432, Z -8.0000, A 0.000, B 0.000, C 0.000 }
gfCNCPoint6[7554] = {X 302.9087, Y 8.8718, Z -8.0000, A 0.000, B 0.000, C 0.000 }
gfCNCPoint6[7555] = {X 303.7126, Y 8.3667, Z -8.0000, A 0.000, B 0.000, C 0.000 }
gfCNCPoint6[7556] = {X 304.6088, Y 8.0531, Z -8.0000, A 0.000, B 0.000, C 0.000 }
gfCNCPoint6[7557] = {X 305.5523, Y 7.9468, Z -8.0000, A 0.000, B 0.000, C 0.000 }
gfCNCPoint6[7558] = {X 311.9957, Y 7.9468, Z -8.0000, A 0.000, B 0.000, C 0.000 }
gfCNCPoint6[7559] = {X 312.9392, Y 8.0531, Z -8.0000, A 0.000, B 0.000, C 0.000 }
gfCNCPoint6[7560] = {X 313.8354, Y 8.3667, Z -8.0000, A 0.000, B 0.000, C 0.000 }
gfCNCPoint6[7561] = {X 314.6393, Y 8.8718, Z -8.0000, A 0.000, B 0.000, C 0.000 }
gfCNCPoint6[7562] = {X 315.3107, Y 9.5432, Z -8.0000, A 0.000, B 0.000, C 0.000 }
gfCNCPoint6[7563] = {X 315.8158, Y 10.3471, Z -8.0000, A 0.000, B 0.000, C 0.000 }
gfCNCPoint6[7564] = {X 316.1294, Y 11.2433, Z -8.0000, A 0.000, B 0.000, C 0.000 }
gfCNCPoint6[7565] = {X 316.2357, Y 12.1868, Z -8.0000, A 0.000, B 0.000, C 0.000 }
gfCNCPoint6[7566] = {X 316.2357, Y 12.9782, Z -8.0000, A 0.000, B 0.000, C 0.000 }
gfCNCPoint6[7567] = {X 316.1344, Y 13.8995, Z -8.0000, A 0.000, B 0.000, C 0.000 }
gfCNCPoint6[7568] = {X 315.8352, Y 14.7769, Z -8.0000, A 0.000, B 0.000, C 0.000 }
gfCNCPoint6[7569] = {X 315.3526, Y 15.5682, Z -8.0000, A 0.000, B 0.000, C 0.000 }
gfCNCPoint6[7570] = {X 314.7095, Y 16.2358, Z -8.0000, A 0.000, B 0.000, C 0.000 }
gfCNCPoint6[7571] = {X 314.7093, Y 40.9516, Z -8.0000, A 0.000, B 0.000, C 0.000 }
gfCNCPoint6[7572] = {X 314.7376, Y 40.9746, Z -8.0000, A 0.000, B 0.000, C 0.000 }
gfCNCPoint6[7573] = {X 315.3637, Y 41.6331, Z -8.0000, A 0.000, B 0.000, C 0.000 }
gfCNCPoint6[7574] = {X 315.8352, Y 42.4099, Z -8.0000, A 0.000, B 0.000, C 0.000 }
gfCNCPoint6[7575] = {X 316.1303, Y 43.2694, Z -8.0000, A 0.000, B 0.000, C 0.000 }
gfCNCPoint6[7576] = {X 316.2356, Y 44.1720, Z -8.0000, A 0.000, B 0.000, C 0.000 }
gfCNCPoint6[7577] = {X 316.2357, Y 45.0000, Z -8.0000, A 0.000, B 0.000, C 0.000 }
gfCNCPoint6[7578] = {X 316.1294, Y 45.9435, Z -8.0000, A 0.000, B 0.000, C 0.000 }
gfCNCPoint6[7579] = {X 315.8158, Y 46.8397, Z -8.0000, A 0.000, B 0.000, C 0.000 }
gfCNCPoint6[7580] = {X 315.3107, Y 47.6436, Z -8.0000, A 0.000, B 0.000, C 0.000 }
gfCNCPoint6[7581] = {X 314.6393, Y 48.3150, Z -8.0000, A 0.000, B 0.000, C 0.000 }
gfCNCPoint6[7582] = {X 313.8354, Y 48.8201, Z -8.0000, A 0.000, B 0.000, C 0.000 }
gfCNCPoint6[7583] = {X 312.9392, Y 49.1337, Z -8.0000, A 0.000, B 0.000, C 0.000 }
gfCNCPoint6[7584] = {X 311.9957, Y 49.2400, Z -8.0000, A 0.000, B 0.000, C 0.000 }
gfCNCPoint6[7585] = {X 305.5523, Y 49.2400, Z -8.0000, A 0.000, B 0.000, C 0.000 }
gfCNCPoint6[7586] = {X 304.6135, Y 49.1348, Z -8.0000, A 0.000, B 0.000, C 0.000 }
gfCNCPoint6[7587] = {X 303.7214, Y 48.8243, Z -8.0000, A 0.000, B 0.000, C 0.000 }
gfCNCPoint6[7588] = {X 302.9201, Y 48.3241, Z -8.0000, A 0.000, B 0.000, C 0.000 }
gfCNCPoint6[7589] = {X 302.2495, Y 47.6588, Z -8.0000, A 0.000, B 0.000, C 0.000 }
gfCNCPoint6[7590] = {X 301.7428, Y 46.8616, Z -8.0000, A 0.000, B 0.000, C 0.000 }
gfCNCPoint6[7591] = {X 301.4252, Y 45.9720, Z -8.0000, A 0.000, B 0.000, C 0.000 }
gfCNCPoint6[7592] = {X 301.3124, Y 45.0341, Z -8.0000, A 0.000, B 0.000, C 0.000 }
gfCNCPoint6[7593] = {X 301.3123, Y 44.2033, Z -8.0000, A 0.000, B 0.000, C 0.000 }
gfCNCPoint6[7594] = {X 301.4292, Y 43.2746, Z -8.0000, A 0.000, B 0.000, C 0.000 }
gfCNCPoint6[7595] = {X 301.7322, Y 42.3890, Z -8.0000, A 0.000, B 0.000, C 0.000 }
gfCNCPoint6[7596] = {X 302.2085, Y 41.5832, Z -8.0000, A 0.000, B 0.000, C 0.000 }
gfCNCPoint6[7597] = {X 302.8384, Y 40.8909, Z -8.0000, A 0.000, B 0.000, C 0.000 }
gfCNCPoint6[7598] = {X 302.8384, Y 33.9543, Z -8.0000, A 0.000, B 0.000, C 0.000 }
gfCNCPoint6[7599] = {X 293.7754, Y 33.9543, Z -8.0000, A 0.000, B 0.000, C 0.000 }
gfCNCPoint6[7600] = {X 293.7749, Y 40.9385, Z -8.0000, A 0.000, B 0.000, C 0.000 }
gfCNCPoint6[7601] = {X 294.4137, Y 41.6122, Z -8.0000, A 0.000, B 0.000, C 0.000 }
gfCNCPoint6[7602] = {X 294.8943, Y 42.4064, Z -8.0000, A 0.000, B 0.000, C 0.000 }
gfCNCPoint6[7603] = {X 295.1947, Y 43.2848, Z -8.0000, A 0.000, B 0.000, C 0.000 }
gfCNCPoint6[7604] = {X 295.3011, Y 44.2070, Z -8.0000, A 0.000, B 0.000, C 0.000 }
gfCNCPoint6[7605] = {X 295.3011, Y 45.0000, Z -8.0000, A 0.000, B 0.000, C 0.000 }
gfCNCPoint6[7606] = {X 295.1948, Y 45.9435, Z -8.0000, A 0.000, B 0.000, C 0.000 }
gfCNCPoint6[7607] = {X 294.8812, Y 46.8397, Z -8.0000, A 0.000, B 0.000, C 0.000 }
gfCNCPoint6[7608] = {X 294.3761, Y 47.6436, Z -8.0000, A 0.000, B 0.000, C 0.000 }
gfCNCPoint6[7609] = {X 293.7047, Y 48.3150, Z -8.0000, A 0.000, B 0.000, C 0.000 }
gfCNCPoint6[7610] = {X 292.9008, Y 48.8201, Z -8.0000, A 0.000, B 0.000, C 0.000 }
gfCNCPoint6[7611] = {X 292.0046, Y 49.1337, Z -8.0000, A 0.000, B 0.000, C 0.000 }
gfCNCPoint6[7612] = {X 291.0611, Y 49.2400, Z -8.0000, A 0.000, B 0.000, C 0.000 }
gfCNCPoint6[7613] = {X 284.6177, Y 49.2400, Z -8.0000, A 0.000, B 0.000, C 0.000 }
gfCNCPoint6[7614] = {X 283.6790, Y 49.1348, Z -8.0000, A 0.000, B 0.000, C 0.000 }
gfCNCPoint6[7615] = {X 282.7869, Y 48.8244, Z -8.0000, A 0.000, B 0.000, C 0.000 }
gfCNCPoint6[7616] = {X 281.9857, Y 48.3242, Z -8.0000, A 0.000, B 0.000, C 0.000 }
gfCNCPoint6[7617] = {X 281.3150, Y 47.6590, Z -8.0000, A 0.000, B 0.000, C 0.000 }
gfCNCPoint6[7618] = {X 280.8083, Y 46.8619, Z -8.0000, A 0.000, B 0.000, C 0.000 }
gfCNCPoint6[7619] = {X 280.4907, Y 45.9723, Z -8.0000, A 0.000, B 0.000, C 0.000 }
gfCNCPoint6[7620] = {X 280.3778, Y 45.0345, Z -8.0000, A 0.000, B 0.000, C 0.000 }
gfCNCPoint6[7621] = {X 280.3777, Y 44.2078, Z -8.0000, A 0.000, B 0.000, C 0.000 }
gfCNCPoint6[7622] = {X 280.4818, Y 43.2866, Z -8.0000, A 0.000, B 0.000, C 0.000 }
gfCNCPoint6[7623] = {X 280.7817, Y 42.4094, Z -8.0000, A 0.000, B 0.000, C 0.000 }
gfCNCPoint6[7624] = {X 281.2633, Y 41.6173, Z -8.0000, A 0.000, B 0.000, C 0.000 }
gfCNCPoint6[7625] = {X 281.9041, Y 40.9473, Z -8.0000, A 0.000, B 0.000, C 0.000 }
gfCNCPoint6[7626] = {X 281.9042, Y 28.5918, Z -8.0000, A 0.000, B 0.000, C 0.000 }
gfCNCPoint6[7627] = {X 277.9042, Y 28.5918, Z -8.0000, A 0.000, B 0.000, C 0.000 }
gfCNCPoint6[7628] = {X 281.9842, Y 28.5918, Z -8.0000, A 0.000, B 0.000, C 0.000 }
gfCNCPoint6[7629] = {X 281.9843, Y 16.1984, Z -8.0000, A 0.000, B 0.000, C 0.000 }
gfCNCPoint6[7630] = {X 281.3471, Y 15.5488, Z -8.0000, A 0.000, B 0.000, C 0.000 }
gfCNCPoint6[7631] = {X 280.8663, Y 14.7761, Z -8.0000, A 0.000, B 0.000, C 0.000 }
gfCNCPoint6[7632] = {X 280.5651, Y 13.9174, Z -8.0000, A 0.000, B 0.000, C 0.000 }
gfCNCPoint6[7633] = {X 280.4578, Y 13.0137, Z -8.0000, A 0.000, B 0.000, C 0.000 }
gfCNCPoint6[7634] = {X 280.4577, Y 12.1868, Z -8.0000, A 0.000, B 0.000, C 0.000 }
gfCNCPoint6[7635] = {X 280.5620, Y 11.2611, Z -8.0000, A 0.000, B 0.000, C 0.000 }
gfCNCPoint6[7636] = {X 280.8696, Y 10.3819, Z -8.0000, A 0.000, B 0.000, C 0.000 }
gfCNCPoint6[7637] = {X 281.3652, Y 9.5931, Z -8.0000, A 0.000, B 0.000, C 0.000 }
gfCNCPoint6[7638] = {X 282.0240, Y 8.9344, Z -8.0000, A 0.000, B 0.000, C 0.000 }
gfCNCPoint6[7639] = {X 282.8127, Y 8.4388, Z -8.0000, A 0.000, B 0.000, C 0.000 }
gfCNCPoint6[7640] = {X 283.6920, Y 8.1311, Z -8.0000, A 0.000, B 0.000, C 0.000 }
gfCNCPoint6[7641] = {X 284.6177, Y 8.0268, Z -8.0000, A 0.000, B 0.000, C 0.000 }
gfCNCPoint6[7642] = {X 291.0611, Y 8.0268, Z -8.0000, A 0.000, B 0.000, C 0.000 }
gfCNCPoint6[7643] = {X 291.9868, Y 8.1311, Z -8.0000, A 0.000, B 0.000, C 0.000 }
gfCNCPoint6[7644] = {X 292.8661, Y 8.4388, Z -8.0000, A 0.000, B 0.000, C 0.000 }
gfCNCPoint6[7645] = {X 293.6549, Y 8.9344, Z -8.0000, A 0.000, B 0.000, C 0.000 }
gfCNCPoint6[7646] = {X 294.3136, Y 9.5931, Z -8.0000, A 0.000, B 0.000, C 0.000 }
gfCNCPoint6[7647] = {X 294.8092, Y 10.3819, Z -8.0000, A 0.000, B 0.000, C 0.000 }
gfCNCPoint6[7648] = {X 295.1168, Y 11.2611, Z -8.0000, A 0.000, B 0.000, C 0.000 }
gfCNCPoint6[7649] = {X 295.2211, Y 12.1868, Z -8.0000, A 0.000, B 0.000, C 0.000 }
gfCNCPoint6[7650] = {X 295.2211, Y 12.9782, Z -8.0000, A 0.000, B 0.000, C 0.000 }
gfCNCPoint6[7651] = {X 295.1255, Y 13.8648, Z -8.0000, A 0.000, B 0.000, C 0.000 }
gfCNCPoint6[7652] = {X 294.8432, Y 14.7106, Z -8.0000, A 0.000, B 0.000, C 0.000 }
gfCNCPoint6[7653] = {X 294.3870, Y 15.4768, Z -8.0000, A 0.000, B 0.000, C 0.000 }
gfCNCPoint6[7654] = {X 293.7780, Y 16.1283, Z -8.0000, A 0.000, B 0.000, C 0.000 }
gfCNCPoint6[7655] = {X 293.6948, Y 16.1982, Z -8.0000, A 0.000, B 0.000, C 0.000 }
gfCNCPoint6[7656] = {X 293.6957, Y 22.3565, Z -8.0000, A 0.000, B 0.000, C 0.000 }
gfCNCPoint6[7657] = {X 302.9181, Y 22.3565, Z -8.0000, A 0.000, B 0.000, C 0.000 }
gfCNCPoint6[7658] = {X 302.9234, Y 16.2021, Z -8.0000, A 0.000, B 0.000, C 0.000 }
gfCNCPoint6[7659] = {X 302.2845, Y 15.5525, Z -8.0000, A 0.000, B 0.000, C 0.000 }
gfCNCPoint6[7660] = {X 301.8025, Y 14.7793, Z -8.0000, A 0.000, B 0.000, C 0.000 }
gfCNCPoint6[7661] = {X 301.5003, Y 13.9198, Z -8.0000, A 0.000, B 0.000, C 0.000 }
gfCNCPoint6[7662] = {X 301.3924, Y 13.0151, Z -8.0000, A 0.000, B 0.000, C 0.000 }
gfCNCPoint6[7663] = {X 301.3923, Y 12.1868, Z -8.0000, A 0.000, B 0.000, C 0.000 }
gfCNCPoint6[7664] = {X 301.4966, Y 11.2611, Z -8.0000, A 0.000, B 0.000, C 0.000 }
gfCNCPoint6[7665] = {X 301.8042, Y 10.3819, Z -8.0000, A 0.000, B 0.000, C 0.000 }
gfCNCPoint6[7666] = {X 302.2998, Y 9.5931, Z -8.0000, A 0.000, B 0.000, C 0.000 }
gfCNCPoint6[7667] = {X 302.9585, Y 8.9344, Z -8.0000, A 0.000, B 0.000, C 0.000 }
gfCNCPoint6[7668] = {X 303.7473, Y 8.4388, Z -8.0000, A 0.000, B 0.000, C 0.000 }
gfCNCPoint6[7669] = {X 304.6266, Y 8.1311, Z -8.0000, A 0.000, B 0.000, C 0.000 }
gfCNCPoint6[7670] = {X 305.5523, Y 8.0268, Z -8.0000, A 0.000, B 0.000, C 0.000 }
gfCNCPoint6[7671] = {X 311.9957, Y 8.0268, Z -8.0000, A 0.000, B 0.000, C 0.000 }
gfCNCPoint6[7672] = {X 312.9214, Y 8.1311, Z -8.0000, A 0.000, B 0.000, C 0.000 }
gfCNCPoint6[7673] = {X 313.8007, Y 8.4388, Z -8.0000, A 0.000, B 0.000, C 0.000 }
gfCNCPoint6[7674] = {X 314.5894, Y 8.9344, Z -8.0000, A 0.000, B 0.000, C 0.000 }
gfCNCPoint6[7675] = {X 315.2481, Y 9.5931, Z -8.0000, A 0.000, B 0.000, C 0.000 }
gfCNCPoint6[7676] = {X 315.7438, Y 10.3819, Z -8.0000, A 0.000, B 0.000, C 0.000 }
gfCNCPoint6[7677] = {X 316.0514, Y 11.2611, Z -8.0000, A 0.000, B 0.000, C 0.000 }
gfCNCPoint6[7678] = {X 316.1557, Y 12.1868, Z -8.0000, A 0.000, B 0.000, C 0.000 }
gfCNCPoint6[7679] = {X 316.1557, Y 12.9782, Z -8.0000, A 0.000, B 0.000, C 0.000 }
gfCNCPoint6[7680] = {X 316.0542, Y 13.8913, Z -8.0000, A 0.000, B 0.000, C 0.000 }
gfCNCPoint6[7681] = {X 315.7548, Y 14.7598, Z -8.0000, A 0.000, B 0.000, C 0.000 }
gfCNCPoint6[7682] = {X 315.2721, Y 15.5414, Z -8.0000, A 0.000, B 0.000, C 0.000 }
gfCNCPoint6[7683] = {X 314.6295, Y 16.1981, Z -8.0000, A 0.000, B 0.000, C 0.000 }
gfCNCPoint6[7684] = {X 314.6293, Y 40.9897, Z -8.0000, A 0.000, B 0.000, C 0.000 }
gfCNCPoint6[7685] = {X 314.6840, Y 41.0341, Z -8.0000, A 0.000, B 0.000, C 0.000 }
gfCNCPoint6[7686] = {X 315.2991, Y 41.6803, Z -8.0000, A 0.000, B 0.000, C 0.000 }
gfCNCPoint6[7687] = {X 315.7623, Y 42.4428, Z -8.0000, A 0.000, B 0.000, C 0.000 }
gfCNCPoint6[7688] = {X 316.0522, Y 43.2865, Z -8.0000, A 0.000, B 0.000, C 0.000 }
gfCNCPoint6[7689] = {X 316.1556, Y 44.1727, Z -8.0000, A 0.000, B 0.000, C 0.000 }
gfCNCPoint6[7690] = {X 316.1557, Y 45.0000, Z -8.0000, A 0.000, B 0.000, C 0.000 }
gfCNCPoint6[7691] = {X 316.0514, Y 45.9257, Z -8.0000, A 0.000, B 0.000, C 0.000 }
gfCNCPoint6[7692] = {X 315.7438, Y 46.8050, Z -8.0000, A 0.000, B 0.000, C 0.000 }
gfCNCPoint6[7693] = {X 315.2481, Y 47.5937, Z -8.0000, A 0.000, B 0.000, C 0.000 }
gfCNCPoint6[7694] = {X 314.5894, Y 48.2524, Z -8.0000, A 0.000, B 0.000, C 0.000 }
gfCNCPoint6[7695] = {X 313.8007, Y 48.7480, Z -8.0000, A 0.000, B 0.000, C 0.000 }
gfCNCPoint6[7696] = {X 312.9214, Y 49.0557, Z -8.0000, A 0.000, B 0.000, C 0.000 }
gfCNCPoint6[7697] = {X 311.9957, Y 49.1600, Z -8.0000, A 0.000, B 0.000, C 0.000 }
gfCNCPoint6[7698] = {X 305.5523, Y 49.1600, Z -8.0000, A 0.000, B 0.000, C 0.000 }
gfCNCPoint6[7699] = {X 304.6312, Y 49.0568, Z -8.0000, A 0.000, B 0.000, C 0.000 }
gfCNCPoint6[7700] = {X 303.7559, Y 48.7522, Z -8.0000, A 0.000, B 0.000, C 0.000 }
gfCNCPoint6[7701] = {X 302.9698, Y 48.2613, Z -8.0000, A 0.000, B 0.000, C 0.000 }
gfCNCPoint6[7702] = {X 302.3118, Y 47.6087, Z -8.0000, A 0.000, B 0.000, C 0.000 }
gfCNCPoint6[7703] = {X 301.8147, Y 46.8265, Z -8.0000, A 0.000, B 0.000, C 0.000 }
gfCNCPoint6[7704] = {X 301.5030, Y 45.9537, Z -8.0000, A 0.000, B 0.000, C 0.000 }
gfCNCPoint6[7705] = {X 301.3924, Y 45.0335, Z -8.0000, A 0.000, B 0.000, C 0.000 }
gfCNCPoint6[7706] = {X 301.3923, Y 44.2051, Z -8.0000, A 0.000, B 0.000, C 0.000 }
gfCNCPoint6[7707] = {X 301.5092, Y 43.2840, Z -8.0000, A 0.000, B 0.000, C 0.000 }
gfCNCPoint6[7708] = {X 301.8123, Y 42.4063, Z -8.0000, A 0.000, B 0.000, C 0.000 }
gfCNCPoint6[7709] = {X 302.2888, Y 41.6093, Z -8.0000, A 0.000, B 0.000, C 0.000 }
gfCNCPoint6[7710] = {X 302.9184, Y 40.9268, Z -8.0000, A 0.000, B 0.000, C 0.000 }
gfCNCPoint6[7711] = {X 302.9184, Y 33.8743, Z -8.0000, A 0.000, B 0.000, C 0.000 }
gfCNCPoint6[7712] = {X 293.6954, Y 33.8743, Z -8.0000, A 0.000, B 0.000, C 0.000 }
gfCNCPoint6[7713] = {X 293.6949, Y 40.9757, Z -8.0000, A 0.000, B 0.000, C 0.000 }
gfCNCPoint6[7714] = {X 294.3332, Y 41.6387, Z -8.0000, A 0.000, B 0.000, C 0.000 }
gfCNCPoint6[7715] = {X 294.8140, Y 42.4236, Z -8.0000, A 0.000, B 0.000, C 0.000 }
gfCNCPoint6[7716] = {X 295.1147, Y 43.2934, Z -8.0000, A 0.000, B 0.000, C 0.000 }
gfCNCPoint6[7717] = {X 295.2211, Y 44.2076, Z -8.0000, A 0.000, B 0.000, C 0.000 }
gfCNCPoint6[7718] = {X 295.2211, Y 45.0000, Z -8.0000, A 0.000, B 0.000, C 0.000 }
gfCNCPoint6[7719] = {X 295.1168, Y 45.9257, Z -8.0000, A 0.000, B 0.000, C 0.000 }
gfCNCPoint6[7720] = {X 294.8092, Y 46.8050, Z -8.0000, A 0.000, B 0.000, C 0.000 }
gfCNCPoint6[7721] = {X 294.3136, Y 47.5937, Z -8.0000, A 0.000, B 0.000, C 0.000 }
gfCNCPoint6[7722] = {X 293.6549, Y 48.2524, Z -8.0000, A 0.000, B 0.000, C 0.000 }
gfCNCPoint6[7723] = {X 292.8661, Y 48.7480, Z -8.0000, A 0.000, B 0.000, C 0.000 }
gfCNCPoint6[7724] = {X 291.9868, Y 49.0557, Z -8.0000, A 0.000, B 0.000, C 0.000 }
gfCNCPoint6[7725] = {X 291.0611, Y 49.1600, Z -8.0000, A 0.000, B 0.000, C 0.000 }
gfCNCPoint6[7726] = {X 284.6177, Y 49.1600, Z -8.0000, A 0.000, B 0.000, C 0.000 }
gfCNCPoint6[7727] = {X 283.6967, Y 49.0568, Z -8.0000, A 0.000, B 0.000, C 0.000 }
gfCNCPoint6[7728] = {X 282.8214, Y 48.7522, Z -8.0000, A 0.000, B 0.000, C 0.000 }
gfCNCPoint6[7729] = {X 282.0353, Y 48.2615, Z -8.0000, A 0.000, B 0.000, C 0.000 }
gfCNCPoint6[7730] = {X 281.3774, Y 47.6088, Z -8.0000, A 0.000, B 0.000, C 0.000 }
gfCNCPoint6[7731] = {X 280.8802, Y 46.8267, Z -8.0000, A 0.000, B 0.000, C 0.000 }
gfCNCPoint6[7732] = {X 280.5685, Y 45.9540, Z -8.0000, A 0.000, B 0.000, C 0.000 }
gfCNCPoint6[7733] = {X 280.4578, Y 45.0339, Z -8.0000, A 0.000, B 0.000, C 0.000 }
gfCNCPoint6[7734] = {X 280.4577, Y 44.2082, Z -8.0000, A 0.000, B 0.000, C 0.000 }
gfCNCPoint6[7735] = {X 280.5619, Y 43.2951, Z -8.0000, A 0.000, B 0.000, C 0.000 }
gfCNCPoint6[7736] = {X 280.8621, Y 42.4266, Z -8.0000, A 0.000, B 0.000, C 0.000 }
gfCNCPoint6[7737] = {X 281.3438, Y 41.6440, Z -8.0000, A 0.000, B 0.000, C 0.000 }
gfCNCPoint6[7738] = {X 281.9841, Y 40.9848, Z -8.0000, A 0.000, B 0.000, C 0.000 }
gfCNCPoint6[7739] = {X 281.9842, Y 28.5918, Z -8.0000, A 0.000, B 0.000, C 0.000 }
gfCNCPoint6[7740] = {X 277.9842, Y 28.5918, Z -8.0000, A 0.000, B 0.000, C 0.000 }
gfCNCPoint6[7741] = {X 282.0642, Y 28.5918, Z -8.0000, A 0.000, B 0.000, C 0.000 }
gfCNCPoint6[7742] = {X 282.0643, Y 16.1603, Z -8.0000, A 0.000, B 0.000, C 0.000 }
gfCNCPoint6[7743] = {X 281.4275, Y 15.5215, Z -8.0000, A 0.000, B 0.000, C 0.000 }
gfCNCPoint6[7744] = {X 280.9467, Y 14.7585, Z -8.0000, A 0.000, B 0.000, C 0.000 }
gfCNCPoint6[7745] = {X 280.6452, Y 13.9085, Z -8.0000, A 0.000, B 0.000, C 0.000 }
gfCNCPoint6[7746] = {X 280.5378, Y 13.0130, Z -8.0000, A 0.000, B 0.000, C 0.000 }
gfCNCPoint6[7747] = {X 280.5377, Y 12.1868, Z -8.0000, A 0.000, B 0.000, C 0.000 }
gfCNCPoint6[7748] = {X 280.6400, Y 11.2789, Z -8.0000, A 0.000, B 0.000, C 0.000 }
gfCNCPoint6[7749] = {X 280.9417, Y 10.4166, Z -8.0000, A 0.000, B 0.000, C 0.000 }
gfCNCPoint6[7750] = {X 281.4278, Y 9.6430, Z -8.0000, A 0.000, B 0.000, C 0.000 }
gfCNCPoint6[7751] = {X 282.0738, Y 8.9969, Z -8.0000, A 0.000, B 0.000, C 0.000 }
gfCNCPoint6[7752] = {X 282.8474, Y 8.5109, Z -8.0000, A 0.000, B 0.000, C 0.000 }
gfCNCPoint6[7753] = {X 283.7098, Y 8.2091, Z -8.0000, A 0.000, B 0.000, C 0.000 }
gfCNCPoint6[7754] = {X 284.6177, Y 8.1068, Z -8.0000, A 0.000, B 0.000, C 0.000 }
gfCNCPoint6[7755] = {X 291.0611, Y 8.1068, Z -8.0000, A 0.000, B 0.000, C 0.000 }
gfCNCPoint6[7756] = {X 291.9690, Y 8.2091, Z -8.0000, A 0.000, B 0.000, C 0.000 }
gfCNCPoint6[7757] = {X 292.8314, Y 8.5109, Z -8.0000, A 0.000, B 0.000, C 0.000 }
gfCNCPoint6[7758] = {X 293.6050, Y 8.9969, Z -8.0000, A 0.000, B 0.000, C 0.000 }
gfCNCPoint6[7759] = {X 294.2510, Y 9.6430, Z -8.0000, A 0.000, B 0.000, C 0.000 }
gfCNCPoint6[7760] = {X 294.7371, Y 10.4166, Z -8.0000, A 0.000, B 0.000, C 0.000 }
gfCNCPoint6[7761] = {X 295.0388, Y 11.2789, Z -8.0000, A 0.000, B 0.000, C 0.000 }
gfCNCPoint6[7762] = {X 295.1411, Y 12.1868, Z -8.0000, A 0.000, B 0.000, C 0.000 }
gfCNCPoint6[7763] = {X 295.1411, Y 12.9782, Z -8.0000, A 0.000, B 0.000, C 0.000 }
gfCNCPoint6[7764] = {X 295.0474, Y 13.8477, Z -8.0000, A 0.000, B 0.000, C 0.000 }
gfCNCPoint6[7765] = {X 294.7704, Y 14.6773, Z -8.0000, A 0.000, B 0.000, C 0.000 }
gfCNCPoint6[7766] = {X 294.3231, Y 15.4288, Z -8.0000, A 0.000, B 0.000, C 0.000 }
gfCNCPoint6[7767] = {X 293.7258, Y 16.0677, Z -8.0000, A 0.000, B 0.000, C 0.000 }
gfCNCPoint6[7768] = {X 293.6682, Y 16.1164, Z -8.0000, A 0.000, B 0.000, C 0.000 }
gfCNCPoint6[7769] = {X 293.6097, Y 16.1641, Z -8.0000, A 0.000, B 0.000, C 0.000 }
gfCNCPoint6[7770] = {X 293.6148, Y 16.1982, Z -8.0000, A 0.000, B 0.000, C 0.000 }
gfCNCPoint6[7771] = {X 293.6157, Y 22.4365, Z -8.0000, A 0.000, B 0.000, C 0.000 }
gfCNCPoint6[7772] = {X 302.9980, Y 22.4365, Z -8.0000, A 0.000, B 0.000, C 0.000 }
gfCNCPoint6[7773] = {X 303.0034, Y 16.1639, Z -8.0000, A 0.000, B 0.000, C 0.000 }
gfCNCPoint6[7774] = {X 302.9449, Y 16.1162, Z -8.0000, A 0.000, B 0.000, C 0.000 }
gfCNCPoint6[7775] = {X 302.8872, Y 16.0674, Z -8.0000, A 0.000, B 0.000, C 0.000 }
gfCNCPoint6[7776] = {X 302.2956, Y 15.4357, Z -8.0000, A 0.000, B 0.000, C 0.000 }
gfCNCPoint6[7777] = {X 301.8504, Y 14.6935, Z -8.0000, A 0.000, B 0.000, C 0.000 }
gfCNCPoint6[7778] = {X 301.5719, Y 13.8741, Z -8.0000, A 0.000, B 0.000, C 0.000 }
gfCNCPoint6[7779] = {X 301.4724, Y 13.0144, Z -8.0000, A 0.000, B 0.000, C 0.000 }
gfCNCPoint6[7780] = {X 301.4723, Y 12.1868, Z -8.0000, A 0.000, B 0.000, C 0.000 }
gfCNCPoint6[7781] = {X 301.5745, Y 11.2789, Z -8.0000, A 0.000, B 0.000, C 0.000 }
gfCNCPoint6[7782] = {X 301.8763, Y 10.4166, Z -8.0000, A 0.000, B 0.000, C 0.000 }
gfCNCPoint6[7783] = {X 302.3624, Y 9.6430, Z -8.0000, A 0.000, B 0.000, C 0.000 }
gfCNCPoint6[7784] = {X 303.0084, Y 8.9969, Z -8.0000, A 0.000, B 0.000, C 0.000 }
gfCNCPoint6[7785] = {X 303.7820, Y 8.5109, Z -8.0000, A 0.000, B 0.000, C 0.000 }
gfCNCPoint6[7786] = {X 304.6444, Y 8.2091, Z -8.0000, A 0.000, B 0.000, C 0.000 }
gfCNCPoint6[7787] = {X 305.5523, Y 8.1068, Z -8.0000, A 0.000, B 0.000, C 0.000 }
gfCNCPoint6[7788] = {X 311.9957, Y 8.1068, Z -8.0000, A 0.000, B 0.000, C 0.000 }
gfCNCPoint6[7789] = {X 312.9036, Y 8.2091, Z -8.0000, A 0.000, B 0.000, C 0.000 }
gfCNCPoint6[7790] = {X 313.7660, Y 8.5109, Z -8.0000, A 0.000, B 0.000, C 0.000 }
gfCNCPoint6[7791] = {X 314.5396, Y 8.9969, Z -8.0000, A 0.000, B 0.000, C 0.000 }
gfCNCPoint6[7792] = {X 315.1856, Y 9.6430, Z -8.0000, A 0.000, B 0.000, C 0.000 }
gfCNCPoint6[7793] = {X 315.6717, Y 10.4166, Z -8.0000, A 0.000, B 0.000, C 0.000 }
gfCNCPoint6[7794] = {X 315.9734, Y 11.2789, Z -8.0000, A 0.000, B 0.000, C 0.000 }
gfCNCPoint6[7795] = {X 316.0757, Y 12.1868, Z -8.0000, A 0.000, B 0.000, C 0.000 }
gfCNCPoint6[7796] = {X 316.0757, Y 12.9782, Z -8.0000, A 0.000, B 0.000, C 0.000 }
gfCNCPoint6[7797] = {X 315.9741, Y 13.8829, Z -8.0000, A 0.000, B 0.000, C 0.000 }
gfCNCPoint6[7798] = {X 315.6744, Y 14.7426, Z -8.0000, A 0.000, B 0.000, C 0.000 }
gfCNCPoint6[7799] = {X 315.1915, Y 15.5144, Z -8.0000, A 0.000, B 0.000, C 0.000 }
gfCNCPoint6[7800] = {X 314.5495, Y 16.1599, Z -8.0000, A 0.000, B 0.000, C 0.000 }
gfCNCPoint6[7801] = {X 314.5493, Y 41.0278, Z -8.0000, A 0.000, B 0.000, C 0.000 }
gfCNCPoint6[7802] = {X 314.6336, Y 41.0962, Z -8.0000, A 0.000, B 0.000, C 0.000 }
gfCNCPoint6[7803] = {X 315.2363, Y 41.7299, Z -8.0000, A 0.000, B 0.000, C 0.000 }
gfCNCPoint6[7804] = {X 315.6902, Y 42.4775, Z -8.0000, A 0.000, B 0.000, C 0.000 }
gfCNCPoint6[7805] = {X 315.9743, Y 43.3047, Z -8.0000, A 0.000, B 0.000, C 0.000 }
gfCNCPoint6[7806] = {X 316.0756, Y 44.1734, Z -8.0000, A 0.000, B 0.000, C 0.000 }
gfCNCPoint6[7807] = {X 316.0757, Y 45.0000, Z -8.0000, A 0.000, B 0.000, C 0.000 }
gfCNCPoint6[7808] = {X 315.9734, Y 45.9079, Z -8.0000, A 0.000, B 0.000, C 0.000 }
gfCNCPoint6[7809] = {X 315.6717, Y 46.7702, Z -8.0000, A 0.000, B 0.000, C 0.000 }
gfCNCPoint6[7810] = {X 315.1856, Y 47.5438, Z -8.0000, A 0.000, B 0.000, C 0.000 }
gfCNCPoint6[7811] = {X 314.5396, Y 48.1899, Z -8.0000, A 0.000, B 0.000, C 0.000 }
gfCNCPoint6[7812] = {X 313.7660, Y 48.6760, Z -8.0000, A 0.000, B 0.000, C 0.000 }
gfCNCPoint6[7813] = {X 312.9036, Y 48.9777, Z -8.0000, A 0.000, B 0.000, C 0.000 }
gfCNCPoint6[7814] = {X 311.9957, Y 49.0800, Z -8.0000, A 0.000, B 0.000, C 0.000 }
gfCNCPoint6[7815] = {X 305.5523, Y 49.0800, Z -8.0000, A 0.000, B 0.000, C 0.000 }
gfCNCPoint6[7816] = {X 304.6489, Y 48.9787, Z -8.0000, A 0.000, B 0.000, C 0.000 }
gfCNCPoint6[7817] = {X 303.7905, Y 48.6800, Z -8.0000, A 0.000, B 0.000, C 0.000 }
gfCNCPoint6[7818] = {X 303.0194, Y 48.1986, Z -8.0000, A 0.000, B 0.000, C 0.000 }
gfCNCPoint6[7819] = {X 302.3741, Y 47.5585, Z -8.0000, A 0.000, B 0.000, C 0.000 }
gfCNCPoint6[7820] = {X 301.8865, Y 46.7914, Z -8.0000, A 0.000, B 0.000, C 0.000 }
gfCNCPoint6[7821] = {X 301.5809, Y 45.9353, Z -8.0000, A 0.000, B 0.000, C 0.000 }
gfCNCPoint6[7822] = {X 301.4724, Y 45.0328, Z -8.0000, A 0.000, B 0.000, C 0.000 }
gfCNCPoint6[7823] = {X 301.4723, Y 44.2070, Z -8.0000, A 0.000, B 0.000, C 0.000 }
gfCNCPoint6[7824] = {X 301.5892, Y 43.2934, Z -8.0000, A 0.000, B 0.000, C 0.000 }
gfCNCPoint6[7825] = {X 301.8925, Y 42.4238, Z -8.0000, A 0.000, B 0.000, C 0.000 }
gfCNCPoint6[7826] = {X 302.3691, Y 41.6356, Z -8.0000, A 0.000, B 0.000, C 0.000 }
gfCNCPoint6[7827] = {X 302.9984, Y 40.9631, Z -8.0000, A 0.000, B 0.000, C 0.000 }
gfCNCPoint6[7828] = {X 302.9984, Y 33.7943, Z -8.0000, A 0.000, B 0.000, C 0.000 }
gfCNCPoint6[7829] = {X 293.6154, Y 33.7943, Z -8.0000, A 0.000, B 0.000, C 0.000 }
gfCNCPoint6[7830] = {X 293.6149, Y 41.0134, Z -8.0000, A 0.000, B 0.000, C 0.000 }
gfCNCPoint6[7831] = {X 294.2528, Y 41.6656, Z -8.0000, A 0.000, B 0.000, C 0.000 }
gfCNCPoint6[7832] = {X 294.7337, Y 42.4409, Z -8.0000, A 0.000, B 0.000, C 0.000 }
gfCNCPoint6[7833] = {X 295.0346, Y 43.3022, Z -8.0000, A 0.000, B 0.000, C 0.000 }
gfCNCPoint6[7834] = {X 295.1411, Y 44.2082, Z -8.0000, A 0.000, B 0.000, C 0.000 }
gfCNCPoint6[7835] = {X 295.1411, Y 45.0000, Z -8.0000, A 0.000, B 0.000, C 0.000 }
gfCNCPoint6[7836] = {X 295.0388, Y 45.9079, Z -8.0000, A 0.000, B 0.000, C 0.000 }
gfCNCPoint6[7837] = {X 294.7371, Y 46.7702, Z -8.0000, A 0.000, B 0.000, C 0.000 }
gfCNCPoint6[7838] = {X 294.2510, Y 47.5438, Z -8.0000, A 0.000, B 0.000, C 0.000 }
gfCNCPoint6[7839] = {X 293.6050, Y 48.1899, Z -8.0000, A 0.000, B 0.000, C 0.000 }
gfCNCPoint6[7840] = {X 292.8314, Y 48.6760, Z -8.0000, A 0.000, B 0.000, C 0.000 }
gfCNCPoint6[7841] = {X 291.9690, Y 48.9777, Z -8.0000, A 0.000, B 0.000, C 0.000 }
gfCNCPoint6[7842] = {X 291.0611, Y 49.0800, Z -8.0000, A 0.000, B 0.000, C 0.000 }
gfCNCPoint6[7843] = {X 284.6177, Y 49.0800, Z -8.0000, A 0.000, B 0.000, C 0.000 }
gfCNCPoint6[7844] = {X 283.7144, Y 48.9788, Z -8.0000, A 0.000, B 0.000, C 0.000 }
gfCNCPoint6[7845] = {X 282.8560, Y 48.6801, Z -8.0000, A 0.000, B 0.000, C 0.000 }
gfCNCPoint6[7846] = {X 282.0850, Y 48.1987, Z -8.0000, A 0.000, B 0.000, C 0.000 }
gfCNCPoint6[7847] = {X 281.4397, Y 47.5587, Z -8.0000, A 0.000, B 0.000, C 0.000 }
gfCNCPoint6[7848] = {X 280.9521, Y 46.7916, Z -8.0000, A 0.000, B 0.000, C 0.000 }
gfCNCPoint6[7849] = {X 280.6464, Y 45.9356, Z -8.0000, A 0.000, B 0.000, C 0.000 }
gfCNCPoint6[7850] = {X 280.5378, Y 45.0332, Z -8.0000, A 0.000, B 0.000, C 0.000 }
gfCNCPoint6[7851] = {X 280.5377, Y 44.2085, Z -8.0000, A 0.000, B 0.000, C 0.000 }
gfCNCPoint6[7852] = {X 280.6420, Y 43.3037, Z -8.0000, A 0.000, B 0.000, C 0.000 }
gfCNCPoint6[7853] = {X 280.9424, Y 42.4439, Z -8.0000, A 0.000, B 0.000, C 0.000 }
gfCNCPoint6[7854] = {X 281.4243, Y 41.6710, Z -8.0000, A 0.000, B 0.000, C 0.000 }
gfCNCPoint6[7855] = {X 282.0641, Y 41.0227, Z -8.0000, A 0.000, B 0.000, C 0.000 }
gfCNCPoint6[7856] = {X 282.0642, Y 28.5918, Z -8.0000, A 0.000, B 0.000, C 0.000 }
gfCNCPoint6[7857] = {X 278.0642, Y 28.5918, Z -8.0000, A 0.000, B 0.000, C 0.000 }
gfCNCPoint6[7858] = {X 282.1442, Y 28.5918, Z -8.0000, A 0.000, B 0.000, C 0.000 }
gfCNCPoint6[7859] = {X 282.1443, Y 16.1216, Z -8.0000, A 0.000, B 0.000, C 0.000 }
gfCNCPoint6[7860] = {X 281.5026, Y 15.4873, Z -8.0000, A 0.000, B 0.000, C 0.000 }
gfCNCPoint6[7861] = {X 281.0195, Y 14.7254, Z -8.0000, A 0.000, B 0.000, C 0.000 }
gfCNCPoint6[7862] = {X 280.7194, Y 13.8745, Z -8.0000, A 0.000, B 0.000, C 0.000 }
gfCNCPoint6[7863] = {X 280.6177, Y 12.9780, Z -8.0000, A 0.000, B 0.000, C 0.000 }
gfCNCPoint6[7864] = {X 280.6177, Y 12.1868, Z -8.0000, A 0.000, B 0.000, C 0.000 }
gfCNCPoint6[7865] = {X 280.7180, Y 11.2967, Z -8.0000, A 0.000, B 0.000, C 0.000 }
gfCNCPoint6[7866] = {X 281.0138, Y 10.4513, Z -8.0000, A 0.000, B 0.000, C 0.000 }
gfCNCPoint6[7867] = {X 281.4903, Y 9.6929, Z -8.0000, A 0.000, B 0.000, C 0.000 }
gfCNCPoint6[7868] = {X 282.1237, Y 9.0595, Z -8.0000, A 0.000, B 0.000, C 0.000 }
gfCNCPoint6[7869] = {X 282.8821, Y 8.5829, Z -8.0000, A 0.000, B 0.000, C 0.000 }
gfCNCPoint6[7870] = {X 283.7276, Y 8.2871, Z -8.0000, A 0.000, B 0.000, C 0.000 }
gfCNCPoint6[7871] = {X 284.6177, Y 8.1868, Z -8.0000, A 0.000, B 0.000, C 0.000 }
gfCNCPoint6[7872] = {X 291.0611, Y 8.1868, Z -8.0000, A 0.000, B 0.000, C 0.000 }
gfCNCPoint6[7873] = {X 291.9512, Y 8.2871, Z -8.0000, A 0.000, B 0.000, C 0.000 }
gfCNCPoint6[7874] = {X 292.7967, Y 8.5829, Z -8.0000, A 0.000, B 0.000, C 0.000 }
gfCNCPoint6[7875] = {X 293.5551, Y 9.0595, Z -8.0000, A 0.000, B 0.000, C 0.000 }
gfCNCPoint6[7876] = {X 294.1885, Y 9.6929, Z -8.0000, A 0.000, B 0.000, C 0.000 }
gfCNCPoint6[7877] = {X 294.6650, Y 10.4513, Z -8.0000, A 0.000, B 0.000, C 0.000 }
gfCNCPoint6[7878] = {X 294.9608, Y 11.2967, Z -8.0000, A 0.000, B 0.000, C 0.000 }
gfCNCPoint6[7879] = {X 295.0611, Y 12.1868, Z -8.0000, A 0.000, B 0.000, C 0.000 }
gfCNCPoint6[7880] = {X 295.0609, Y 13.0192, Z -8.0000, A 0.000, B 0.000, C 0.000 }
gfCNCPoint6[7881] = {X 294.9625, Y 13.8607, Z -8.0000, A 0.000, B 0.000, C 0.000 }
gfCNCPoint6[7882] = {X 294.6891, Y 14.6626, Z -8.0000, A 0.000, B 0.000, C 0.000 }
gfCNCPoint6[7883] = {X 294.2529, Y 15.3889, Z -8.0000, A 0.000, B 0.000, C 0.000 }
gfCNCPoint6[7884] = {X 293.6736, Y 16.0071, Z -8.0000, A 0.000, B 0.000, C 0.000 }
gfCNCPoint6[7885] = {X 293.5964, Y 16.0719, Z -8.0000, A 0.000, B 0.000, C 0.000 }
gfCNCPoint6[7886] = {X 293.5177, Y 16.1348, Z -8.0000, A 0.000, B 0.000, C 0.000 }
gfCNCPoint6[7887] = {X 293.5348, Y 16.1929, Z -8.0000, A 0.000, B 0.000, C 0.000 }
gfCNCPoint6[7888] = {X 293.5349, Y 16.7687, Z -8.0000, A 0.000, B 0.000, C 0.000 }
gfCNCPoint6[7889] = {X 293.5357, Y 22.5165, Z -8.0000, A 0.000, B 0.000, C 0.000 }
gfCNCPoint6[7890] = {X 303.0780, Y 22.5165, Z -8.0000, A 0.000, B 0.000, C 0.000 }
gfCNCPoint6[7891] = {X 303.0782, Y 16.1930, Z -8.0000, A 0.000, B 0.000, C 0.000 }
gfCNCPoint6[7892] = {X 303.0955, Y 16.1346, Z -8.0000, A 0.000, B 0.000, C 0.000 }
gfCNCPoint6[7893] = {X 303.0167, Y 16.0717, Z -8.0000, A 0.000, B 0.000, C 0.000 }
gfCNCPoint6[7894] = {X 302.9395, Y 16.0068, Z -8.0000, A 0.000, B 0.000, C 0.000 }
gfCNCPoint6[7895] = {X 302.3541, Y 15.3804, Z -8.0000, A 0.000, B 0.000, C 0.000 }
gfCNCPoint6[7896] = {X 301.9156, Y 14.6437, Z -8.0000, A 0.000, B 0.000, C 0.000 }
gfCNCPoint6[7897] = {X 301.6441, Y 13.8304, Z -8.0000, A 0.000, B 0.000, C 0.000 }
gfCNCPoint6[7898] = {X 301.5523, Y 12.9780, Z -8.0000, A 0.000, B 0.000, C 0.000 }
gfCNCPoint6[7899] = {X 301.5523, Y 12.1868, Z -8.0000, A 0.000, B 0.000, C 0.000 }
gfCNCPoint6[7900] = {X 301.6525, Y 11.2967, Z -8.0000, A 0.000, B 0.000, C 0.000 }
gfCNCPoint6[7901] = {X 301.9484, Y 10.4513, Z -8.0000, A 0.000, B 0.000, C 0.000 }
gfCNCPoint6[7902] = {X 302.4249, Y 9.6929, Z -8.0000, A 0.000, B 0.000, C 0.000 }
gfCNCPoint6[7903] = {X 303.0583, Y 9.0595, Z -8.0000, A 0.000, B 0.000, C 0.000 }
gfCNCPoint6[7904] = {X 303.8167, Y 8.5829, Z -8.0000, A 0.000, B 0.000, C 0.000 }
gfCNCPoint6[7905] = {X 304.6622, Y 8.2871, Z -8.0000, A 0.000, B 0.000, C 0.000 }
gfCNCPoint6[7906] = {X 305.5523, Y 8.1868, Z -8.0000, A 0.000, B 0.000, C 0.000 }
gfCNCPoint6[7907] = {X 311.9957, Y 8.1868, Z -8.0000, A 0.000, B 0.000, C 0.000 }
gfCNCPoint6[7908] = {X 312.8858, Y 8.2871, Z -8.0000, A 0.000, B 0.000, C 0.000 }
gfCNCPoint6[7909] = {X 313.7313, Y 8.5829, Z -8.0000, A 0.000, B 0.000, C 0.000 }
gfCNCPoint6[7910] = {X 314.4897, Y 9.0595, Z -8.0000, A 0.000, B 0.000, C 0.000 }
gfCNCPoint6[7911] = {X 315.1230, Y 9.6929, Z -8.0000, A 0.000, B 0.000, C 0.000 }
gfCNCPoint6[7912] = {X 315.5996, Y 10.4513, Z -8.0000, A 0.000, B 0.000, C 0.000 }
gfCNCPoint6[7913] = {X 315.8954, Y 11.2967, Z -8.0000, A 0.000, B 0.000, C 0.000 }
gfCNCPoint6[7914] = {X 315.9957, Y 12.1868, Z -8.0000, A 0.000, B 0.000, C 0.000 }
gfCNCPoint6[7915] = {X 315.9955, Y 13.0192, Z -8.0000, A 0.000, B 0.000, C 0.000 }
gfCNCPoint6[7916] = {X 315.8870, Y 13.9044, Z -8.0000, A 0.000, B 0.000, C 0.000 }
gfCNCPoint6[7917] = {X 315.5850, Y 14.7436, Z -8.0000, A 0.000, B 0.000, C 0.000 }
gfCNCPoint6[7918] = {X 315.1045, Y 15.4950, Z -8.0000, A 0.000, B 0.000, C 0.000 }
gfCNCPoint6[7919] = {X 314.4695, Y 16.1213, Z -8.0000, A 0.000, B 0.000, C 0.000 }
gfCNCPoint6[7920] = {X 314.4693, Y 41.0659, Z -8.0000, A 0.000, B 0.000, C 0.000 }
gfCNCPoint6[7921] = {X 314.6081, Y 41.1797, Z -8.0000, A 0.000, B 0.000, C 0.000 }
gfCNCPoint6[7922] = {X 315.1937, Y 41.8061, Z -8.0000, A 0.000, B 0.000, C 0.000 }
gfCNCPoint6[7923] = {X 315.6323, Y 42.5429, Z -8.0000, A 0.000, B 0.000, C 0.000 }
gfCNCPoint6[7924] = {X 315.9038, Y 43.3563, Z -8.0000, A 0.000, B 0.000, C 0.000 }
gfCNCPoint6[7925] = {X 315.9957, Y 44.2089, Z -8.0000, A 0.000, B 0.000, C 0.000 }
gfCNCPoint6[7926] = {X 315.9957, Y 45.0000, Z -8.0000, A 0.000, B 0.000, C 0.000 }
gfCNCPoint6[7927] = {X 315.8954, Y 45.8901, Z -8.0000, A 0.000, B 0.000, C 0.000 }
gfCNCPoint6[7928] = {X 315.5996, Y 46.7355, Z -8.0000, A 0.000, B 0.000, C 0.000 }
gfCNCPoint6[7929] = {X 315.1230, Y 47.4940, Z -8.0000, A 0.000, B 0.000, C 0.000 }
gfCNCPoint6[7930] = {X 314.4897, Y 48.1273, Z -8.0000, A 0.000, B 0.000, C 0.000 }
gfCNCPoint6[7931] = {X 313.7313, Y 48.6039, Z -8.0000, A 0.000, B 0.000, C 0.000 }
gfCNCPoint6[7932] = {X 312.8858, Y 48.8997, Z -8.0000, A 0.000, B 0.000, C 0.000 }
gfCNCPoint6[7933] = {X 311.9957, Y 49.0000, Z -8.0000, A 0.000, B 0.000, C 0.000 }
gfCNCPoint6[7934] = {X 305.5523, Y 49.0000, Z -8.0000, A 0.000, B 0.000, C 0.000 }
gfCNCPoint6[7935] = {X 304.6622, Y 48.8997, Z -8.0000, A 0.000, B 0.000, C 0.000 }
gfCNCPoint6[7936] = {X 303.8167, Y 48.6039, Z -8.0000, A 0.000, B 0.000, C 0.000 }
gfCNCPoint6[7937] = {X 303.0583, Y 48.1273, Z -8.0000, A 0.000, B 0.000, C 0.000 }
gfCNCPoint6[7938] = {X 302.4249, Y 47.4939, Z -8.0000, A 0.000, B 0.000, C 0.000 }
gfCNCPoint6[7939] = {X 301.9484, Y 46.7355, Z -8.0000, A 0.000, B 0.000, C 0.000 }
gfCNCPoint6[7940] = {X 301.6525, Y 45.8901, Z -8.0000, A 0.000, B 0.000, C 0.000 }
gfCNCPoint6[7941] = {X 301.5523, Y 45.0000, Z -8.0000, A 0.000, B 0.000, C 0.000 }
gfCNCPoint6[7942] = {X 301.5523, Y 44.2088, Z -8.0000, A 0.000, B 0.000, C 0.000 }
gfCNCPoint6[7943] = {X 301.6691, Y 43.3029, Z -8.0000, A 0.000, B 0.000, C 0.000 }
gfCNCPoint6[7944] = {X 301.9726, Y 42.4414, Z -8.0000, A 0.000, B 0.000, C 0.000 }
gfCNCPoint6[7945] = {X 302.4494, Y 41.6622, Z -8.0000, A 0.000, B 0.000, C 0.000 }
gfCNCPoint6[7946] = {X 303.0784, Y 40.9999, Z -8.0000, A 0.000, B 0.000, C 0.000 }
gfCNCPoint6[7947] = {X 303.0784, Y 33.7143, Z -8.0000, A 0.000, B 0.000, C 0.000 }
gfCNCPoint6[7948] = {X 293.5354, Y 33.7143, Z -8.0000, A 0.000, B 0.000, C 0.000 }
gfCNCPoint6[7949] = {X 293.5349, Y 41.0514, Z -8.0000, A 0.000, B 0.000, C 0.000 }
gfCNCPoint6[7950] = {X 294.1723, Y 41.6928, Z -8.0000, A 0.000, B 0.000, C 0.000 }
gfCNCPoint6[7951] = {X 294.6533, Y 42.4584, Z -8.0000, A 0.000, B 0.000, C 0.000 }
gfCNCPoint6[7952] = {X 294.9545, Y 43.3110, Z -8.0000, A 0.000, B 0.000, C 0.000 }
gfCNCPoint6[7953] = {X 295.0611, Y 44.2088, Z -8.0000, A 0.000, B 0.000, C 0.000 }
gfCNCPoint6[7954] = {X 295.0611, Y 45.0000, Z -8.0000, A 0.000, B 0.000, C 0.000 }
gfCNCPoint6[7955] = {X 294.9608, Y 45.8901, Z -8.0000, A 0.000, B 0.000, C 0.000 }
gfCNCPoint6[7956] = {X 294.6650, Y 46.7355, Z -8.0000, A 0.000, B 0.000, C 0.000 }
gfCNCPoint6[7957] = {X 294.1885, Y 47.4940, Z -8.0000, A 0.000, B 0.000, C 0.000 }
gfCNCPoint6[7958] = {X 293.5551, Y 48.1273, Z -8.0000, A 0.000, B 0.000, C 0.000 }
gfCNCPoint6[7959] = {X 292.7967, Y 48.6039, Z -8.0000, A 0.000, B 0.000, C 0.000 }
gfCNCPoint6[7960] = {X 291.9512, Y 48.8997, Z -8.0000, A 0.000, B 0.000, C 0.000 }
gfCNCPoint6[7961] = {X 291.0611, Y 49.0000, Z -8.0000, A 0.000, B 0.000, C 0.000 }
gfCNCPoint6[7962] = {X 284.6177, Y 49.0000, Z -8.0000, A 0.000, B 0.000, C 0.000 }
gfCNCPoint6[7963] = {X 283.7276, Y 48.8997, Z -8.0000, A 0.000, B 0.000, C 0.000 }
gfCNCPoint6[7964] = {X 282.8821, Y 48.6039, Z -8.0000, A 0.000, B 0.000, C 0.000 }
gfCNCPoint6[7965] = {X 282.1237, Y 48.1273, Z -8.0000, A 0.000, B 0.000, C 0.000 }
gfCNCPoint6[7966] = {X 281.4903, Y 47.4939, Z -8.0000, A 0.000, B 0.000, C 0.000 }
gfCNCPoint6[7967] = {X 281.0138, Y 46.7355, Z -8.0000, A 0.000, B 0.000, C 0.000 }
gfCNCPoint6[7968] = {X 280.7180, Y 45.8901, Z -8.0000, A 0.000, B 0.000, C 0.000 }
gfCNCPoint6[7969] = {X 280.6177, Y 45.0000, Z -8.0000, A 0.000, B 0.000, C 0.000 }
gfCNCPoint6[7970] = {X 280.6177, Y 44.2088, Z -8.0000, A 0.000, B 0.000, C 0.000 }
gfCNCPoint6[7971] = {X 280.7221, Y 43.3123, Z -8.0000, A 0.000, B 0.000, C 0.000 }
gfCNCPoint6[7972] = {X 281.0228, Y 42.4613, Z -8.0000, A 0.000, B 0.000, C 0.000 }
gfCNCPoint6[7973] = {X 281.5048, Y 41.6982, Z -8.0000, A 0.000, B 0.000, C 0.000 }
gfCNCPoint6[7974] = {X 282.1441, Y 41.0611, Z -8.0000, A 0.000, B 0.000, C 0.000 }
gfCNCPoint6[7975] = {X 282.1442, Y 28.5918, Z -8.0000, A 0.000, B 0.000, C 0.000 }
gfCNCPoint6[7976] = {X 278.0642, Y 28.5918, Z -8.0000, A 0.000, B 0.000, C 0.000 }
gfCNCPoint6[7977] = {X 278.0642, Y 28.5918, Z -5.0000, A 0.000, B 0.000, C 0.000 }
gfCNCPoint6[7978] = {X 278.0642, Y 28.5918, Z 11.0000, A 0.000, B 0.000, C 0.000 }
gfCNCPoint6[7979] = {X 349.6581, Y 107.1078, Z 11.0000, A 0.000, B 0.000, C 0.000 }
gfCNCPoint6[7980] = {X 349.6581, Y 107.1078, Z -5.0000, A 0.000, B 0.000, C 0.000 }
gfCNCPoint6[7981] = {X 349.6581, Y 107.1078, Z -8.0000, A 0.000, B 0.000, C 0.000 }
gfCNCPoint6[7982] = {X 349.6273, Y 103.0279, Z -8.0000, A 0.000, B 0.000, C 0.000 }
gfCNCPoint6[7983] = {X 345.9299, Y 103.0183, Z -8.0000, A 0.000, B 0.000, C 0.000 }
gfCNCPoint6[7984] = {X 342.2334, Y 102.9335, Z -8.0000, A 0.000, B 0.000, C 0.000 }
gfCNCPoint6[7985] = {X 337.5902, Y 102.7434, Z -8.0000, A 0.000, B 0.000, C 0.000 }
gfCNCPoint6[7986] = {X 332.9586, Y 102.3634, Z -8.0000, A 0.000, B 0.000, C 0.000 }
gfCNCPoint6[7987] = {X 328.3465, Y 101.7942, Z -8.0000, A 0.000, B 0.000, C 0.000 }
gfCNCPoint6[7988] = {X 325.2777, Y 101.2557, Z -8.0000, A 0.000, B 0.000, C 0.000 }
gfCNCPoint6[7989] = {X 322.2519, Y 100.5122, Z -8.0000, A 0.000, B 0.000, C 0.000 }
gfCNCPoint6[7990] = {X 319.2829, Y 99.5671, Z -8.0000, A 0.000, B 0.000, C 0.000 }
gfCNCPoint6[7991] = {X 317.5439, Y 98.8715, Z -8.0000, A 0.000, B 0.000, C 0.000 }
gfCNCPoint6[7992] = {X 315.8700, Y 98.0313, Z -8.0000, A 0.000, B 0.000, C 0.000 }
gfCNCPoint6[7993] = {X 314.2732, Y 97.0526, Z -8.0000, A 0.000, B 0.000, C 0.000 }
gfCNCPoint6[7994] = {X 312.7648, Y 95.9424, Z -8.0000, A 0.000, B 0.000, C 0.000 }
gfCNCPoint6[7995] = {X 311.6085, Y 94.8855, Z -8.0000, A 0.000, B 0.000, C 0.000 }
gfCNCPoint6[7996] = {X 310.5963, Y 93.6898, Z -8.0000, A 0.000, B 0.000, C 0.000 }
gfCNCPoint6[7997] = {X 309.7447, Y 92.3749, Z -8.0000, A 0.000, B 0.000, C 0.000 }
gfCNCPoint6[7998] = {X 309.0675, Y 90.9623, Z -8.0000, A 0.000, B 0.000, C 0.000 }
gfCNCPoint6[7999] = {X 308.5012, Y 89.1237, Z -8.0000, A 0.000, B 0.000, C 0.000 }
gfCNCPoint6[8000] = {X 308.1464, Y 87.2329, Z -8.0000, A 0.000, B 0.000, C 0.000 }
gfCNCPoint6[8001] = {X 308.0076, Y 85.3141, Z -8.0000, A 0.000, B 0.000, C 0.000 }
gfCNCPoint6[8002] = {X 307.9940, Y 84.6190, Z -8.0000, A 0.000, B 0.000, C 0.000 }
gfCNCPoint6[8003] = {X 307.9953, Y 63.2121, Z -8.0000, A 0.000, B 0.000, C 0.000 }
gfCNCPoint6[8004] = {X 307.1440, Y 63.0027, Z -8.0000, A 0.000, B 0.000, C 0.000 }
gfCNCPoint6[8005] = {X 306.3525, Y 62.6257, Z -8.0000, A 0.000, B 0.000, C 0.000 }
gfCNCPoint6[8006] = {X 305.6534, Y 62.0967, Z -8.0000, A 0.000, B 0.000, C 0.000 }
gfCNCPoint6[8007] = {X 305.0755, Y 61.4375, Z -8.0000, A 0.000, B 0.000, C 0.000 }
gfCNCPoint6[8008] = {X 304.6426, Y 60.6752, Z -8.0000, A 0.000, B 0.000, C 0.000 }
gfCNCPoint6[8009] = {X 304.3725, Y 59.8411, Z -8.0000, A 0.000, B 0.000, C 0.000 }
gfCNCPoint6[8010] = {X 304.2764, Y 58.9697, Z -8.0000, A 0.000, B 0.000, C 0.000 }
gfCNCPoint6[8011] = {X 304.2762, Y 58.0000, Z -8.0000, A 0.000, B 0.000, C 0.000 }
gfCNCPoint6[8012] = {X 304.3845, Y 57.0387, Z -8.0000, A 0.000, B 0.000, C 0.000 }
gfCNCPoint6[8013] = {X 304.7040, Y 56.1256, Z -8.0000, A 0.000, B 0.000, C 0.000 }
gfCNCPoint6[8014] = {X 305.2187, Y 55.3065, Z -8.0000, A 0.000, B 0.000, C 0.000 }
gfCNCPoint6[8015] = {X 305.9027, Y 54.6225, Z -8.0000, A 0.000, B 0.000, C 0.000 }
gfCNCPoint6[8016] = {X 306.7218, Y 54.1078, Z -8.0000, A 0.000, B 0.000, C 0.000 }
gfCNCPoint6[8017] = {X 307.6349, Y 53.7883, Z -8.0000, A 0.000, B 0.000, C 0.000 }
gfCNCPoint6[8018] = {X 308.5962, Y 53.6800, Z -8.0000, A 0.000, B 0.000, C 0.000 }
gfCNCPoint6[8019] = {X 324.3107, Y 53.6800, Z -8.0000, A 0.000, B 0.000, C 0.000 }
gfCNCPoint6[8020] = {X 325.2720, Y 53.7883, Z -8.0000, A 0.000, B 0.000, C 0.000 }
gfCNCPoint6[8021] = {X 326.1851, Y 54.1078, Z -8.0000, A 0.000, B 0.000, C 0.000 }
gfCNCPoint6[8022] = {X 327.0042, Y 54.6225, Z -8.0000, A 0.000, B 0.000, C 0.000 }
gfCNCPoint6[8023] = {X 327.6882, Y 55.3065, Z -8.0000, A 0.000, B 0.000, C 0.000 }
gfCNCPoint6[8024] = {X 328.2029, Y 56.1256, Z -8.0000, A 0.000, B 0.000, C 0.000 }
gfCNCPoint6[8025] = {X 328.5224, Y 57.0387, Z -8.0000, A 0.000, B 0.000, C 0.000 }
gfCNCPoint6[8026] = {X 328.6307, Y 58.0000, Z -8.0000, A 0.000, B 0.000, C 0.000 }
gfCNCPoint6[8027] = {X 328.6307, Y 58.9357, Z -8.0000, A 0.000, B 0.000, C 0.000 }
gfCNCPoint6[8028] = {X 328.5370, Y 59.8122, Z -8.0000, A 0.000, B 0.000, C 0.000 }
gfCNCPoint6[8029] = {X 328.2689, Y 60.6518, Z -8.0000, A 0.000, B 0.000, C 0.000 }
gfCNCPoint6[8030] = {X 327.8373, Y 61.4203, Z -8.0000, A 0.000, B 0.000, C 0.000 }
gfCNCPoint6[8031] = {X 327.2598, Y 62.0862, Z -8.0000, A 0.000, B 0.000, C 0.000 }
gfCNCPoint6[8032] = {X 326.5602, Y 62.6222, Z -8.0000, A 0.000, B 0.000, C 0.000 }
gfCNCPoint6[8033] = {X 325.7669, Y 63.0065, Z -8.0000, A 0.000, B 0.000, C 0.000 }
gfCNCPoint6[8034] = {X 324.9126, Y 63.2232, Z -8.0000, A 0.000, B 0.000, C 0.000 }
gfCNCPoint6[8035] = {X 324.9146, Y 83.2296, Z -8.0000, A 0.000, B 0.000, C 0.000 }
gfCNCPoint6[8036] = {X 324.9281, Y 84.6145, Z -8.0000, A 0.000, B 0.000, C 0.000 }
gfCNCPoint6[8037] = {X 325.0048, Y 85.8429, Z -8.0000, A 0.000, B 0.000, C 0.000 }
gfCNCPoint6[8038] = {X 325.2231, Y 87.0541, Z -8.0000, A 0.000, B 0.000, C 0.000 }
gfCNCPoint6[8039] = {X 325.6727, Y 87.4781, Z -8.0000, A 0.000, B 0.000, C 0.000 }
gfCNCPoint6[8040] = {X 326.2087, Y 87.7855, Z -8.0000, A 0.000, B 0.000, C 0.000 }
gfCNCPoint6[8041] = {X 327.9884, Y 88.4968, Z -8.0000, A 0.000, B 0.000, C 0.000 }
gfCNCPoint6[8042] = {X 329.8404, Y 88.9897, Z -8.0000, A 0.000, B 0.000, C 0.000 }
gfCNCPoint6[8043] = {X 332.9244, Y 89.5430, Z -8.0000, A 0.000, B 0.000, C 0.000 }
gfCNCPoint6[8044] = {X 336.0365, Y 89.9074, Z -8.0000, A 0.000, B 0.000, C 0.000 }
gfCNCPoint6[8045] = {X 340.4062, Y 90.2016, Z -8.0000, A 0.000, B 0.000, C 0.000 }
gfCNCPoint6[8046] = {X 344.7832, Y 90.3554, Z -8.0000, A 0.000, B 0.000, C 0.000 }
gfCNCPoint6[8047] = {X 349.1628, Y 90.3687, Z -8.0000, A 0.000, B 0.000, C 0.000 }
gfCNCPoint6[8048] = {X 353.3143, Y 90.3004, Z -8.0000, A 0.000, B 0.000, C 0.000 }
gfCNCPoint6[8049] = {X 357.4607, Y 90.0814, Z -8.0000, A 0.000, B 0.000, C 0.000 }
gfCNCPoint6[8050] = {X 361.5963, Y 89.7120, Z -8.0000, A 0.000, B 0.000, C 0.000 }
gfCNCPoint6[8051] = {X 363.6775, Y 89.4249, Z -8.0000, A 0.000, B 0.000, C 0.000 }
gfCNCPoint6[8052] = {X 365.7397, Y 89.0229, Z -8.0000, A 0.000, B 0.000, C 0.000 }
gfCNCPoint6[8053] = {X 367.7763, Y 88.5073, Z -8.0000, A 0.000, B 0.000, C 0.000 }
gfCNCPoint6[8054] = {X 368.7087, Y 88.1943, Z -8.0000, A 0.000, B 0.000, C 0.000 }
gfCNCPoint6[8055] = {X 369.5999, Y 87.7784, Z -8.0000, A 0.000, B 0.000, C 0.000 }
gfCNCPoint6[8056] = {X 370.4386, Y 87.2648, Z -8.0000, A 0.000, B 0.000, C 0.000 }
gfCNCPoint6[8057] = {X 370.5871, Y 87.1101, Z -8.0000, A 0.000, B 0.000, C 0.000 }
gfCNCPoint6[8058] = {X 370.6637, Y 86.9097, Z -8.0000, A 0.000, B 0.000, C 0.000 }
gfCNCPoint6[8059] = {X 370.8549, Y 85.3747, Z -8.0000, A 0.000, B 0.000, C 0.000 }
gfCNCPoint6[8060] = {X 370.9187, Y 83.8290, Z -8.0000, A 0.000, B 0.000, C 0.000 }
gfCNCPoint6[8061] = {X 370.9198, Y 63.2123, Z -8.0000, A 0.000, B 0.000, C 0.000 }
gfCNCPoint6[8062] = {X 370.0682, Y 63.0031, Z -8.0000, A 0.000, B 0.000, C 0.000 }
gfCNCPoint6[8063] = {X 369.2765, Y 62.6262, Z -8.0000, A 0.000, B 0.000, C 0.000 }
gfCNCPoint6[8064] = {X 368.5771, Y 62.0973, Z -8.0000, A 0.000, B 0.000, C 0.000 }
gfCNCPoint6[8065] = {X 367.9989, Y 61.4380, Z -8.0000, A 0.000, B 0.000, C 0.000 }
gfCNCPoint6[8066] = {X 367.5658, Y 60.6755, Z -8.0000, A 0.000, B 0.000, C 0.000 }
gfCNCPoint6[8067] = {X 367.2956, Y 59.8413, Z -8.0000, A 0.000, B 0.000, C 0.000 }
gfCNCPoint6[8068] = {X 367.1994, Y 58.9697, Z -8.0000, A 0.000, B 0.000, C 0.000 }
gfCNCPoint6[8069] = {X 367.1993, Y 58.0000, Z -8.0000, A 0.000, B 0.000, C 0.000 }
gfCNCPoint6[8070] = {X 367.3076, Y 57.0387, Z -8.0000, A 0.000, B 0.000, C 0.000 }
gfCNCPoint6[8071] = {X 367.6271, Y 56.1256, Z -8.0000, A 0.000, B 0.000, C 0.000 }
gfCNCPoint6[8072] = {X 368.1418, Y 55.3065, Z -8.0000, A 0.000, B 0.000, C 0.000 }
gfCNCPoint6[8073] = {X 368.8258, Y 54.6225, Z -8.0000, A 0.000, B 0.000, C 0.000 }
gfCNCPoint6[8074] = {X 369.6449, Y 54.1078, Z -8.0000, A 0.000, B 0.000, C 0.000 }
gfCNCPoint6[8075] = {X 370.5580, Y 53.7883, Z -8.0000, A 0.000, B 0.000, C 0.000 }
gfCNCPoint6[8076] = {X 371.5193, Y 53.6800, Z -8.0000, A 0.000, B 0.000, C 0.000 }
gfCNCPoint6[8077] = {X 388.0597, Y 53.6800, Z -8.0000, A 0.000, B 0.000, C 0.000 }
gfCNCPoint6[8078] = {X 389.0210, Y 53.7883, Z -8.0000, A 0.000, B 0.000, C 0.000 }
gfCNCPoint6[8079] = {X 389.9341, Y 54.1078, Z -8.0000, A 0.000, B 0.000, C 0.000 }
gfCNCPoint6[8080] = {X 390.7532, Y 54.6225, Z -8.0000, A 0.000, B 0.000, C 0.000 }
gfCNCPoint6[8081] = {X 391.4372, Y 55.3065, Z -8.0000, A 0.000, B 0.000, C 0.000 }
gfCNCPoint6[8082] = {X 391.9519, Y 56.1256, Z -8.0000, A 0.000, B 0.000, C 0.000 }
gfCNCPoint6[8083] = {X 392.2714, Y 57.0387, Z -8.0000, A 0.000, B 0.000, C 0.000 }
gfCNCPoint6[8084] = {X 392.3797, Y 58.0000, Z -8.0000, A 0.000, B 0.000, C 0.000 }
gfCNCPoint6[8085] = {X 392.3797, Y 58.9342, Z -8.0000, A 0.000, B 0.000, C 0.000 }
gfCNCPoint6[8086] = {X 392.2728, Y 59.8892, Z -8.0000, A 0.000, B 0.000, C 0.000 }
gfCNCPoint6[8087] = {X 391.9574, Y 60.7969, Z -8.0000, A 0.000, B 0.000, C 0.000 }
gfCNCPoint6[8088] = {X 391.5173, Y 61.5258, Z -8.0000, A 0.000, B 0.000, C 0.000 }
gfCNCPoint6[8089] = {X 390.9434, Y 62.1549, Z -8.0000, A 0.000, B 0.000, C 0.000 }
gfCNCPoint6[8090] = {X 390.2579, Y 62.6599, Z -8.0000, A 0.000, B 0.000, C 0.000 }
gfCNCPoint6[8091] = {X 389.4869, Y 63.0215, Z -8.0000, A 0.000, B 0.000, C 0.000 }
gfCNCPoint6[8092] = {X 388.6603, Y 63.2257, Z -8.0000, A 0.000, B 0.000, C 0.000 }
gfCNCPoint6[8093] = {X 388.6583, Y 84.6147, Z -8.0000, A 0.000, B 0.000, C 0.000 }
gfCNCPoint6[8094] = {X 388.5984, Y 86.2730, Z -8.0000, A 0.000, B 0.000, C 0.000 }
gfCNCPoint6[8095] = {X 388.3940, Y 87.9198, Z -8.0000, A 0.000, B 0.000, C 0.000 }
gfCNCPoint6[8096] = {X 388.0468, Y 89.5425, Z -8.0000, A 0.000, B 0.000, C 0.000 }
gfCNCPoint6[8097] = {X 387.5177, Y 91.1213, Z -8.0000, A 0.000, B 0.000, C 0.000 }
gfCNCPoint6[8098] = {X 386.7737, Y 92.6109, Z -8.0000, A 0.000, B 0.000, C 0.000 }
gfCNCPoint6[8099] = {X 385.8294, Y 93.9823, Z -8.0000, A 0.000, B 0.000, C 0.000 }
gfCNCPoint6[8100] = {X 384.7030, Y 95.2086, Z -8.0000, A 0.000, B 0.000, C 0.000 }
gfCNCPoint6[8101] = {X 383.1818, Y 96.4964, Z -8.0000, A 0.000, B 0.000, C 0.000 }
gfCNCPoint6[8102] = {X 381.5311, Y 97.6135, Z -8.0000, A 0.000, B 0.000, C 0.000 }
gfCNCPoint6[8103] = {X 379.7701, Y 98.5470, Z -8.0000, A 0.000, B 0.000, C 0.000 }
gfCNCPoint6[8104] = {X 377.4987, Y 99.5019, Z -8.0000, A 0.000, B 0.000, C 0.000 }
gfCNCPoint6[8105] = {X 375.1648, Y 100.2921, Z -8.0000, A 0.000, B 0.000, C 0.000 }
gfCNCPoint6[8106] = {X 372.7804, Y 100.9136, Z -8.0000, A 0.000, B 0.000, C 0.000 }
gfCNCPoint6[8107] = {X 369.0988, Y 101.6300, Z -8.0000, A 0.000, B 0.000, C 0.000 }
gfCNCPoint6[8108] = {X 365.3875, Y 102.1722, Z -8.0000, A 0.000, B 0.000, C 0.000 }
gfCNCPoint6[8109] = {X 361.6549, Y 102.5389, Z -8.0000, A 0.000, B 0.000, C 0.000 }
gfCNCPoint6[8110] = {X 355.6451, Y 102.8829, Z -8.0000, A 0.000, B 0.000, C 0.000 }
gfCNCPoint6[8111] = {X 349.6273, Y 103.0279, Z -8.0000, A 0.000, B 0.000, C 0.000 }
gfCNCPoint6[8112] = {X 349.6575, Y 107.0278, Z -8.0000, A 0.000, B 0.000, C 0.000 }
gfCNCPoint6[8113] = {X 349.6267, Y 102.9479, Z -8.0000, A 0.000, B 0.000, C 0.000 }
gfCNCPoint6[8114] = {X 345.9306, Y 102.9383, Z -8.0000, A 0.000, B 0.000, C 0.000 }
gfCNCPoint6[8115] = {X 342.2356, Y 102.8536, Z -8.0000, A 0.000, B 0.000, C 0.000 }
gfCNCPoint6[8116] = {X 337.5954, Y 102.6635, Z -8.0000, A 0.000, B 0.000, C 0.000 }
gfCNCPoint6[8117] = {X 332.9669, Y 102.2838, Z -8.0000, A 0.000, B 0.000, C 0.000 }
gfCNCPoint6[8118] = {X 328.3579, Y 101.7150, Z -8.0000, A 0.000, B 0.000, C 0.000 }
gfCNCPoint6[8119] = {X 325.2942, Y 101.1774, Z -8.0000, A 0.000, B 0.000, C 0.000 }
gfCNCPoint6[8120] = {X 322.2735, Y 100.4351, Z -8.0000, A 0.000, B 0.000, C 0.000 }
gfCNCPoint6[8121] = {X 319.3096, Y 99.4916, Z -8.0000, A 0.000, B 0.000, C 0.000 }
gfCNCPoint6[8122] = {X 317.5769, Y 98.7986, Z -8.0000, A 0.000, B 0.000, C 0.000 }
gfCNCPoint6[8123] = {X 315.9090, Y 97.9614, Z -8.0000, A 0.000, B 0.000, C 0.000 }
gfCNCPoint6[8124] = {X 314.3178, Y 96.9863, Z -8.0000, A 0.000, B 0.000, C 0.000 }
gfCNCPoint6[8125] = {X 312.8149, Y 95.8801, Z -8.0000, A 0.000, B 0.000, C 0.000 }
gfCNCPoint6[8126] = {X 311.6663, Y 94.8302, Z -8.0000, A 0.000, B 0.000, C 0.000 }
gfCNCPoint6[8127] = {X 310.6609, Y 93.6426, Z -8.0000, A 0.000, B 0.000, C 0.000 }
gfCNCPoint6[8128] = {X 309.8149, Y 92.3366, Z -8.0000, A 0.000, B 0.000, C 0.000 }
gfCNCPoint6[8129] = {X 309.1421, Y 90.9334, Z -8.0000, A 0.000, B 0.000, C 0.000 }
gfCNCPoint6[8130] = {X 308.5786, Y 89.1037, Z -8.0000, A 0.000, B 0.000, C 0.000 }
gfCNCPoint6[8131] = {X 308.2256, Y 87.2221, Z -8.0000, A 0.000, B 0.000, C 0.000 }
gfCNCPoint6[8132] = {X 308.0876, Y 85.3126, Z -8.0000, A 0.000, B 0.000, C 0.000 }
gfCNCPoint6[8133] = {X 308.0740, Y 84.6182, Z -8.0000, A 0.000, B 0.000, C 0.000 }
gfCNCPoint6[8134] = {X 308.0753, Y 63.1419, Z -8.0000, A 0.000, B 0.000, C 0.000 }
gfCNCPoint6[8135] = {X 307.2271, Y 62.9469, Z -8.0000, A 0.000, B 0.000, C 0.000 }
gfCNCPoint6[8136] = {X 306.4366, Y 62.5829, Z -8.0000, A 0.000, B 0.000, C 0.000 }
gfCNCPoint6[8137] = {X 305.7371, Y 62.0651, Z -8.0000, A 0.000, B 0.000, C 0.000 }
gfCNCPoint6[8138] = {X 305.1581, Y 61.4153, Z -8.0000, A 0.000, B 0.000, C 0.000 }
gfCNCPoint6[8139] = {X 304.7239, Y 60.6611, Z -8.0000, A 0.000, B 0.000, C 0.000 }
gfCNCPoint6[8140] = {X 304.4528, Y 59.8340, Z -8.0000, A 0.000, B 0.000, C 0.000 }
gfCNCPoint6[8141] = {X 304.3564, Y 58.9691, Z -8.0000, A 0.000, B 0.000, C 0.000 }
gfCNCPoint6[8142] = {X 304.3562, Y 58.0000, Z -8.0000, A 0.000, B 0.000, C 0.000 }
gfCNCPoint6[8143] = {X 304.4625, Y 57.0565, Z -8.0000, A 0.000, B 0.000, C 0.000 }
gfCNCPoint6[8144] = {X 304.7761, Y 56.1603, Z -8.0000, A 0.000, B 0.000, C 0.000 }
gfCNCPoint6[8145] = {X 305.2813, Y 55.3564, Z -8.0000, A 0.000, B 0.000, C 0.000 }
gfCNCPoint6[8146] = {X 305.9526, Y 54.6850, Z -8.0000, A 0.000, B 0.000, C 0.000 }
gfCNCPoint6[8147] = {X 306.7566, Y 54.1799, Z -8.0000, A 0.000, B 0.000, C 0.000 }
gfCNCPoint6[8148] = {X 307.6527, Y 53.8663, Z -8.0000, A 0.000, B 0.000, C 0.000 }
gfCNCPoint6[8149] = {X 308.5962, Y 53.7600, Z -8.0000, A 0.000, B 0.000, C 0.000 }
gfCNCPoint6[8150] = {X 324.3107, Y 53.7600, Z -8.0000, A 0.000, B 0.000, C 0.000 }
gfCNCPoint6[8151] = {X 325.2542, Y 53.8663, Z -8.0000, A 0.000, B 0.000, C 0.000 }
gfCNCPoint6[8152] = {X 326.1504, Y 54.1799, Z -8.0000, A 0.000, B 0.000, C 0.000 }
gfCNCPoint6[8153] = {X 326.9543, Y 54.6850, Z -8.0000, A 0.000, B 0.000, C 0.000 }
gfCNCPoint6[8154] = {X 327.6257, Y 55.3564, Z -8.0000, A 0.000, B 0.000, C 0.000 }
gfCNCPoint6[8155] = {X 328.1308, Y 56.1603, Z -8.0000, A 0.000, B 0.000, C 0.000 }
gfCNCPoint6[8156] = {X 328.4444, Y 57.0565, Z -8.0000, A 0.000, B 0.000, C 0.000 }
gfCNCPoint6[8157] = {X 328.5507, Y 58.0000, Z -8.0000, A 0.000, B 0.000, C 0.000 }
gfCNCPoint6[8158] = {X 328.5507, Y 58.9353, Z -8.0000, A 0.000, B 0.000, C 0.000 }
gfCNCPoint6[8159] = {X 328.4567, Y 59.8053, Z -8.0000, A 0.000, B 0.000, C 0.000 }
gfCNCPoint6[8160] = {X 328.1877, Y 60.6379, Z -8.0000, A 0.000, B 0.000, C 0.000 }
gfCNCPoint6[8161] = {X 327.7548, Y 61.3984, Z -8.0000, A 0.000, B 0.000, C 0.000 }
gfCNCPoint6[8162] = {X 327.1762, Y 62.0548, Z -8.0000, A 0.000, B 0.000, C 0.000 }
gfCNCPoint6[8163] = {X 326.4761, Y 62.5797, Z -8.0000, A 0.000, B 0.000, C 0.000 }
gfCNCPoint6[8164] = {X 325.6839, Y 62.9512, Z -8.0000, A 0.000, B 0.000, C 0.000 }
gfCNCPoint6[8165] = {X 324.8326, Y 63.1536, Z -8.0000, A 0.000, B 0.000, C 0.000 }
gfCNCPoint6[8166] = {X 324.8346, Y 83.2300, Z -8.0000, A 0.000, B 0.000, C 0.000 }
gfCNCPoint6[8167] = {X 324.8481, Y 84.6148, Z -8.0000, A 0.000, B 0.000, C 0.000 }
gfCNCPoint6[8168] = {X 324.9265, Y 85.8617, Z -8.0000, A 0.000, B 0.000, C 0.000 }
gfCNCPoint6[8169] = {X 325.1497, Y 87.0910, Z -8.0000, A 0.000, B 0.000, C 0.000 }
gfCNCPoint6[8170] = {X 325.6168, Y 87.5363, Z -8.0000, A 0.000, B 0.000, C 0.000 }
gfCNCPoint6[8171] = {X 326.1760, Y 87.8585, Z -8.0000, A 0.000, B 0.000, C 0.000 }
gfCNCPoint6[8172] = {X 327.9639, Y 88.5730, Z -8.0000, A 0.000, B 0.000, C 0.000 }
gfCNCPoint6[8173] = {X 329.8245, Y 89.0681, Z -8.0000, A 0.000, B 0.000, C 0.000 }
gfCNCPoint6[8174] = {X 332.9131, Y 89.6222, Z -8.0000, A 0.000, B 0.000, C 0.000 }
gfCNCPoint6[8175] = {X 336.0297, Y 89.9871, Z -8.0000, A 0.000, B 0.000, C 0.000 }
gfCNCPoint6[8176] = {X 340.4020, Y 90.2815, Z -8.0000, A 0.000, B 0.000, C 0.000 }
gfCNCPoint6[8177] = {X 344.7816, Y 90.4354, Z -8.0000, A 0.000, B 0.000, C 0.000 }
gfCNCPoint6[8178] = {X 349.1638, Y 90.4487, Z -8.0000, A 0.000, B 0.000, C 0.000 }
gfCNCPoint6[8179] = {X 353.3179, Y 90.3803, Z -8.0000, A 0.000, B 0.000, C 0.000 }
gfCNCPoint6[8180] = {X 357.4668, Y 90.1611, Z -8.0000, A 0.000, B 0.000, C 0.000 }
gfCNCPoint6[8181] = {X 361.6051, Y 89.7915, Z -8.0000, A 0.000, B 0.000, C 0.000 }
gfCNCPoint6[8182] = {X 363.6907, Y 89.5039, Z -8.0000, A 0.000, B 0.000, C 0.000 }
gfCNCPoint6[8183] = {X 365.7571, Y 89.1010, Z -8.0000, A 0.000, B 0.000, C 0.000 }
gfCNCPoint6[8184] = {X 367.7981, Y 88.5843, Z -8.0000, A 0.000, B 0.000, C 0.000 }
gfCNCPoint6[8185] = {X 368.7388, Y 88.2685, Z -8.0000, A 0.000, B 0.000, C 0.000 }
gfCNCPoint6[8186] = {X 369.6379, Y 87.8488, Z -8.0000, A 0.000, B 0.000, C 0.000 }
gfCNCPoint6[8187] = {X 370.4841, Y 87.3306, Z -8.0000, A 0.000, B 0.000, C 0.000 }
gfCNCPoint6[8188] = {X 370.6547, Y 87.1529, Z -8.0000, A 0.000, B 0.000, C 0.000 }
gfCNCPoint6[8189] = {X 370.7426, Y 86.9229, Z -8.0000, A 0.000, B 0.000, C 0.000 }
gfCNCPoint6[8190] = {X 370.9346, Y 85.3813, Z -8.0000, A 0.000, B 0.000, C 0.000 }
gfCNCPoint6[8191] = {X 370.9987, Y 83.8290, Z -8.0000, A 0.000, B 0.000, C 0.000 }
gfCNCPoint6[8192] = {X 370.9998, Y 63.1421, Z -8.0000, A 0.000, B 0.000, C 0.000 }
gfCNCPoint6[8193] = {X 370.1514, Y 62.9473, Z -8.0000, A 0.000, B 0.000, C 0.000 }
gfCNCPoint6[8194] = {X 369.3606, Y 62.5834, Z -8.0000, A 0.000, B 0.000, C 0.000 }
gfCNCPoint6[8195] = {X 368.6608, Y 62.0656, Z -8.0000, A 0.000, B 0.000, C 0.000 }
gfCNCPoint6[8196] = {X 368.0815, Y 61.4158, Z -8.0000, A 0.000, B 0.000, C 0.000 }
gfCNCPoint6[8197] = {X 367.6471, Y 60.6614, Z -8.0000, A 0.000, B 0.000, C 0.000 }
gfCNCPoint6[8198] = {X 367.3759, Y 59.8342, Z -8.0000, A 0.000, B 0.000, C 0.000 }
gfCNCPoint6[8199] = {X 367.2794, Y 58.9691, Z -8.0000, A 0.000, B 0.000, C 0.000 }
gfCNCPoint6[8200] = {X 367.2793, Y 58.0000, Z -8.0000, A 0.000, B 0.000, C 0.000 }
gfCNCPoint6[8201] = {X 367.3856, Y 57.0565, Z -8.0000, A 0.000, B 0.000, C 0.000 }
gfCNCPoint6[8202] = {X 367.6992, Y 56.1603, Z -8.0000, A 0.000, B 0.000, C 0.000 }
gfCNCPoint6[8203] = {X 368.2043, Y 55.3564, Z -8.0000, A 0.000, B 0.000, C 0.000 }
gfCNCPoint6[8204] = {X 368.8757, Y 54.6850, Z -8.0000, A 0.000, B 0.000, C 0.000 }
gfCNCPoint6[8205] = {X 369.6796, Y 54.1799, Z -8.0000, A 0.000, B 0.000, C 0.000 }
gfCNCPoint6[8206] = {X 370.5758, Y 53.8663, Z -8.0000, A 0.000, B 0.000, C 0.000 }
gfCNCPoint6[8207] = {X 371.5193, Y 53.7600, Z -8.0000, A 0.000, B 0.000, C 0.000 }
gfCNCPoint6[8208] = {X 388.0597, Y 53.7600, Z -8.0000, A 0.000, B 0.000, C 0.000 }
gfCNCPoint6[8209] = {X 389.0032, Y 53.8663, Z -8.0000, A 0.000, B 0.000, C 0.000 }
gfCNCPoint6[8210] = {X 389.8993, Y 54.1799, Z -8.0000, A 0.000, B 0.000, C 0.000 }
gfCNCPoint6[8211] = {X 390.7033, Y 54.6850, Z -8.0000, A 0.000, B 0.000, C 0.000 }
gfCNCPoint6[8212] = {X 391.3746, Y 55.3564, Z -8.0000, A 0.000, B 0.000, C 0.000 }
gfCNCPoint6[8213] = {X 391.8798, Y 56.1603, Z -8.0000, A 0.000, B 0.000, C 0.000 }
gfCNCPoint6[8214] = {X 392.1934, Y 57.0565, Z -8.0000, A 0.000, B 0.000, C 0.000 }
gfCNCPoint6[8215] = {X 392.2997, Y 58.0000, Z -8.0000, A 0.000, B 0.000, C 0.000 }
gfCNCPoint6[8216] = {X 392.2997, Y 58.9342, Z -8.0000, A 0.000, B 0.000, C 0.000 }
gfCNCPoint6[8217] = {X 392.1948, Y 59.8715, Z -8.0000, A 0.000, B 0.000, C 0.000 }
gfCNCPoint6[8218] = {X 391.8852, Y 60.7624, Z -8.0000, A 0.000, B 0.000, C 0.000 }
gfCNCPoint6[8219] = {X 391.4449, Y 61.4890, Z -8.0000, A 0.000, B 0.000, C 0.000 }
gfCNCPoint6[8220] = {X 390.8693, Y 62.1138, Z -8.0000, A 0.000, B 0.000, C 0.000 }
gfCNCPoint6[8221] = {X 390.1812, Y 62.6122, Z -8.0000, A 0.000, B 0.000, C 0.000 }
gfCNCPoint6[8222] = {X 389.4080, Y 62.9642, Z -8.0000, A 0.000, B 0.000, C 0.000 }
gfCNCPoint6[8223] = {X 388.5803, Y 63.1559, Z -8.0000, A 0.000, B 0.000, C 0.000 }
gfCNCPoint6[8224] = {X 388.5783, Y 84.6150, Z -8.0000, A 0.000, B 0.000, C 0.000 }
gfCNCPoint6[8225] = {X 388.5186, Y 86.2665, Z -8.0000, A 0.000, B 0.000, C 0.000 }
gfCNCPoint6[8226] = {X 388.3151, Y 87.9065, Z -8.0000, A 0.000, B 0.000, C 0.000 }
gfCNCPoint6[8227] = {X 387.9694, Y 89.5225, Z -8.0000, A 0.000, B 0.000, C 0.000 }
gfCNCPoint6[8228] = {X 387.4438, Y 91.0906, Z -8.0000, A 0.000, B 0.000, C 0.000 }
gfCNCPoint6[8229] = {X 386.7048, Y 92.5703, Z -8.0000, A 0.000, B 0.000, C 0.000 }
gfCNCPoint6[8230] = {X 385.7668, Y 93.9324, Z -8.0000, A 0.000, B 0.000, C 0.000 }
gfCNCPoint6[8231] = {X 384.6480, Y 95.1505, Z -8.0000, A 0.000, B 0.000, C 0.000 }
gfCNCPoint6[8232] = {X 383.1334, Y 96.4327, Z -8.0000, A 0.000, B 0.000, C 0.000 }
gfCNCPoint6[8233] = {X 381.4899, Y 97.5449, Z -8.0000, A 0.000, B 0.000, C 0.000 }
gfCNCPoint6[8234] = {X 379.7365, Y 98.4744, Z -8.0000, A 0.000, B 0.000, C 0.000 }
gfCNCPoint6[8235] = {X 377.4703, Y 99.4271, Z -8.0000, A 0.000, B 0.000, C 0.000 }
gfCNCPoint6[8236] = {X 375.1418, Y 100.2155, Z -8.0000, A 0.000, B 0.000, C 0.000 }
gfCNCPoint6[8237] = {X 372.7630, Y 100.8355, Z -8.0000, A 0.000, B 0.000, C 0.000 }
gfCNCPoint6[8238] = {X 369.0852, Y 101.5511, Z -8.0000, A 0.000, B 0.000, C 0.000 }
gfCNCPoint6[8239] = {X 365.3777, Y 102.0928, Z -8.0000, A 0.000, B 0.000, C 0.000 }
gfCNCPoint6[8240] = {X 361.6489, Y 102.4591, Z -8.0000, A 0.000, B 0.000, C 0.000 }
gfCNCPoint6[8241] = {X 355.6418, Y 102.8029, Z -8.0000, A 0.000, B 0.000, C 0.000 }
gfCNCPoint6[8242] = {X 349.6267, Y 102.9479, Z -8.0000, A 0.000, B 0.000, C 0.000 }
gfCNCPoint6[8243] = {X 349.6569, Y 106.9478, Z -8.0000, A 0.000, B 0.000, C 0.000 }
gfCNCPoint6[8244] = {X 349.6261, Y 102.8679, Z -8.0000, A 0.000, B 0.000, C 0.000 }
gfCNCPoint6[8245] = {X 345.9314, Y 102.8583, Z -8.0000, A 0.000, B 0.000, C 0.000 }
gfCNCPoint6[8246] = {X 342.2377, Y 102.7736, Z -8.0000, A 0.000, B 0.000, C 0.000 }
gfCNCPoint6[8247] = {X 337.6007, Y 102.5837, Z -8.0000, A 0.000, B 0.000, C 0.000 }
gfCNCPoint6[8248] = {X 332.9752, Y 102.2042, Z -8.0000, A 0.000, B 0.000, C 0.000 }
gfCNCPoint6[8249] = {X 328.3692, Y 101.6358, Z -8.0000, A 0.000, B 0.000, C 0.000 }
gfCNCPoint6[8250] = {X 325.3107, Y 101.0991, Z -8.0000, A 0.000, B 0.000, C 0.000 }
gfCNCPoint6[8251] = {X 322.2952, Y 100.3581, Z -8.0000, A 0.000, B 0.000, C 0.000 }
gfCNCPoint6[8252] = {X 319.3362, Y 99.4162, Z -8.0000, A 0.000, B 0.000, C 0.000 }
gfCNCPoint6[8253] = {X 317.6098, Y 98.7256, Z -8.0000, A 0.000, B 0.000, C 0.000 }
gfCNCPoint6[8254] = {X 315.9479, Y 97.8916, Z -8.0000, A 0.000, B 0.000, C 0.000 }
gfCNCPoint6[8255] = {X 314.3625, Y 96.9199, Z -8.0000, A 0.000, B 0.000, C 0.000 }
gfCNCPoint6[8256] = {X 312.8650, Y 95.8177, Z -8.0000, A 0.000, B 0.000, C 0.000 }
gfCNCPoint6[8257] = {X 311.7242, Y 94.7749, Z -8.0000, A 0.000, B 0.000, C 0.000 }
gfCNCPoint6[8258] = {X 310.7254, Y 93.5953, Z -8.0000, A 0.000, B 0.000, C 0.000 }
gfCNCPoint6[8259] = {X 309.8851, Y 92.2982, Z -8.0000, A 0.000, B 0.000, C 0.000 }
gfCNCPoint6[8260] = {X 309.2168, Y 90.9045, Z -8.0000, A 0.000, B 0.000, C 0.000 }
gfCNCPoint6[8261] = {X 308.6561, Y 89.0838, Z -8.0000, A 0.000, B 0.000, C 0.000 }
gfCNCPoint6[8262] = {X 308.3049, Y 87.2113, Z -8.0000, A 0.000, B 0.000, C 0.000 }
gfCNCPoint6[8263] = {X 308.1676, Y 85.3111, Z -8.0000, A 0.000, B 0.000, C 0.000 }
gfCNCPoint6[8264] = {X 308.1540, Y 84.6175, Z -8.0000, A 0.000, B 0.000, C 0.000 }
gfCNCPoint6[8265] = {X 308.1553, Y 63.0706, Z -8.0000, A 0.000, B 0.000, C 0.000 }
gfCNCPoint6[8266] = {X 307.3104, Y 62.8904, Z -8.0000, A 0.000, B 0.000, C 0.000 }
gfCNCPoint6[8267] = {X 306.5209, Y 62.5395, Z -8.0000, A 0.000, B 0.000, C 0.000 }
gfCNCPoint6[8268] = {X 305.8210, Y 62.0331, Z -8.0000, A 0.000, B 0.000, C 0.000 }
gfCNCPoint6[8269] = {X 305.2407, Y 61.3930, Z -8.0000, A 0.000, B 0.000, C 0.000 }
gfCNCPoint6[8270] = {X 304.8052, Y 60.6469, Z -8.0000, A 0.000, B 0.000, C 0.000 }
gfCNCPoint6[8271] = {X 304.5332, Y 59.8269, Z -8.0000, A 0.000, B 0.000, C 0.000 }
gfCNCPoint6[8272] = {X 304.4364, Y 58.9684, Z -8.0000, A 0.000, B 0.000, C 0.000 }
gfCNCPoint6[8273] = {X 304.4362, Y 58.0000, Z -8.0000, A 0.000, B 0.000, C 0.000 }
gfCNCPoint6[8274] = {X 304.5405, Y 57.0743, Z -8.0000, A 0.000, B 0.000, C 0.000 }
gfCNCPoint6[8275] = {X 304.8482, Y 56.1950, Z -8.0000, A 0.000, B 0.000, C 0.000 }
gfCNCPoint6[8276] = {X 305.3438, Y 55.4063, Z -8.0000, A 0.000, B 0.000, C 0.000 }
gfCNCPoint6[8277] = {X 306.0025, Y 54.7476, Z -8.0000, A 0.000, B 0.000, C 0.000 }
gfCNCPoint6[8278] = {X 306.7913, Y 54.2520, Z -8.0000, A 0.000, B 0.000, C 0.000 }
gfCNCPoint6[8279] = {X 307.6705, Y 53.9443, Z -8.0000, A 0.000, B 0.000, C 0.000 }
gfCNCPoint6[8280] = {X 308.5962, Y 53.8400, Z -8.0000, A 0.000, B 0.000, C 0.000 }
gfCNCPoint6[8281] = {X 324.3107, Y 53.8400, Z -8.0000, A 0.000, B 0.000, C 0.000 }
gfCNCPoint6[8282] = {X 325.2364, Y 53.9443, Z -8.0000, A 0.000, B 0.000, C 0.000 }
gfCNCPoint6[8283] = {X 326.1156, Y 54.2520, Z -8.0000, A 0.000, B 0.000, C 0.000 }
gfCNCPoint6[8284] = {X 326.9044, Y 54.7476, Z -8.0000, A 0.000, B 0.000, C 0.000 }
gfCNCPoint6[8285] = {X 327.5631, Y 55.4063, Z -8.0000, A 0.000, B 0.000, C 0.000 }
gfCNCPoint6[8286] = {X 328.0587, Y 56.1950, Z -8.0000, A 0.000, B 0.000, C 0.000 }
gfCNCPoint6[8287] = {X 328.3664, Y 57.0743, Z -8.0000, A 0.000, B 0.000, C 0.000 }
gfCNCPoint6[8288] = {X 328.4707, Y 58.0000, Z -8.0000, A 0.000, B 0.000, C 0.000 }
gfCNCPoint6[8289] = {X 328.4707, Y 58.9349, Z -8.0000, A 0.000, B 0.000, C 0.000 }
gfCNCPoint6[8290] = {X 328.3764, Y 59.7984, Z -8.0000, A 0.000, B 0.000, C 0.000 }
gfCNCPoint6[8291] = {X 328.1063, Y 60.6240, Z -8.0000, A 0.000, B 0.000, C 0.000 }
gfCNCPoint6[8292] = {X 327.6721, Y 61.3763, Z -8.0000, A 0.000, B 0.000, C 0.000 }
gfCNCPoint6[8293] = {X 327.0924, Y 62.0231, Z -8.0000, A 0.000, B 0.000, C 0.000 }
gfCNCPoint6[8294] = {X 326.3919, Y 62.5367, Z -8.0000, A 0.000, B 0.000, C 0.000 }
gfCNCPoint6[8295] = {X 325.6006, Y 62.8951, Z -8.0000, A 0.000, B 0.000, C 0.000 }
gfCNCPoint6[8296] = {X 324.7526, Y 63.0829, Z -8.0000, A 0.000, B 0.000, C 0.000 }
gfCNCPoint6[8297] = {X 324.7546, Y 83.2304, Z -8.0000, A 0.000, B 0.000, C 0.000 }
gfCNCPoint6[8298] = {X 324.7681, Y 84.6152, Z -8.0000, A 0.000, B 0.000, C 0.000 }
gfCNCPoint6[8299] = {X 324.8482, Y 85.8805, Z -8.0000, A 0.000, B 0.000, C 0.000 }
gfCNCPoint6[8300] = {X 325.0763, Y 87.1276, Z -8.0000, A 0.000, B 0.000, C 0.000 }
gfCNCPoint6[8301] = {X 325.5609, Y 87.5944, Z -8.0000, A 0.000, B 0.000, C 0.000 }
gfCNCPoint6[8302] = {X 326.1432, Y 87.9315, Z -8.0000, A 0.000, B 0.000, C 0.000 }
gfCNCPoint6[8303] = {X 327.9394, Y 88.6491, Z -8.0000, A 0.000, B 0.000, C 0.000 }
gfCNCPoint6[8304] = {X 329.8086, Y 89.1465, Z -8.0000, A 0.000, B 0.000, C 0.000 }
gfCNCPoint6[8305] = {X 332.9017, Y 89.7014, Z -8.0000, A 0.000, B 0.000, C 0.000 }
gfCNCPoint6[8306] = {X 336.0228, Y 90.0668, Z -8.0000, A 0.000, B 0.000, C 0.000 }
gfCNCPoint6[8307] = {X 340.3978, Y 90.3614, Z -8.0000, A 0.000, B 0.000, C 0.000 }
gfCNCPoint6[8308] = {X 344.7800, Y 90.5154, Z -8.0000, A 0.000, B 0.000, C 0.000 }
gfCNCPoint6[8309] = {X 349.1649, Y 90.5287, Z -8.0000, A 0.000, B 0.000, C 0.000 }
gfCNCPoint6[8310] = {X 353.3215, Y 90.4602, Z -8.0000, A 0.000, B 0.000, C 0.000 }
gfCNCPoint6[8311] = {X 357.4730, Y 90.2409, Z -8.0000, A 0.000, B 0.000, C 0.000 }
gfCNCPoint6[8312] = {X 361.6137, Y 89.8711, Z -8.0000, A 0.000, B 0.000, C 0.000 }
gfCNCPoint6[8313] = {X 363.7037, Y 89.5828, Z -8.0000, A 0.000, B 0.000, C 0.000 }
gfCNCPoint6[8314] = {X 365.7746, Y 89.1791, Z -8.0000, A 0.000, B 0.000, C 0.000 }
gfCNCPoint6[8315] = {X 367.8199, Y 88.6612, Z -8.0000, A 0.000, B 0.000, C 0.000 }
gfCNCPoint6[8316] = {X 368.7689, Y 88.3426, Z -8.0000, A 0.000, B 0.000, C 0.000 }
gfCNCPoint6[8317] = {X 369.6760, Y 87.9191, Z -8.0000, A 0.000, B 0.000, C 0.000 }
gfCNCPoint6[8318] = {X 370.5297, Y 87.3963, Z -8.0000, A 0.000, B 0.000, C 0.000 }
gfCNCPoint6[8319] = {X 370.7222, Y 87.1958, Z -8.0000, A 0.000, B 0.000, C 0.000 }
gfCNCPoint6[8320] = {X 370.8215, Y 86.9361, Z -8.0000, A 0.000, B 0.000, C 0.000 }
gfCNCPoint6[8321] = {X 371.0144, Y 85.3879, Z -8.0000, A 0.000, B 0.000, C 0.000 }
gfCNCPoint6[8322] = {X 371.0787, Y 83.8290, Z -8.0000, A 0.000, B 0.000, C 0.000 }
gfCNCPoint6[8323] = {X 371.0798, Y 63.0708, Z -8.0000, A 0.000, B 0.000, C 0.000 }
gfCNCPoint6[8324] = {X 370.9771, Y 63.0586, Z -8.0000, A 0.000, B 0.000, C 0.000 }
gfCNCPoint6[8325] = {X 370.8748, Y 63.0438, Z -8.0000, A 0.000, B 0.000, C 0.000 }
gfCNCPoint6[8326] = {X 369.9375, Y 62.7816, Z -8.0000, A 0.000, B 0.000, C 0.000 }
gfCNCPoint6[8327] = {X 369.0868, Y 62.3088, Z -8.0000, A 0.000, B 0.000, C 0.000 }
gfCNCPoint6[8328] = {X 368.3693, Y 61.6512, Z -8.0000, A 0.000, B 0.000, C 0.000 }
gfCNCPoint6[8329] = {X 367.8241, Y 60.8449, Z -8.0000, A 0.000, B 0.000, C 0.000 }
gfCNCPoint6[8330] = {X 367.4813, Y 59.9340, Z -8.0000, A 0.000, B 0.000, C 0.000 }
gfCNCPoint6[8331] = {X 367.3594, Y 58.9684, Z -8.0000, A 0.000, B 0.000, C 0.000 }
gfCNCPoint6[8332] = {X 367.3593, Y 58.0000, Z -8.0000, A 0.000, B 0.000, C 0.000 }
gfCNCPoint6[8333] = {X 367.4636, Y 57.0743, Z -8.0000, A 0.000, B 0.000, C 0.000 }
gfCNCPoint6[8334] = {X 367.7713, Y 56.1950, Z -8.0000, A 0.000, B 0.000, C 0.000 }
gfCNCPoint6[8335] = {X 368.2669, Y 55.4063, Z -8.0000, A 0.000, B 0.000, C 0.000 }
gfCNCPoint6[8336] = {X 368.9256, Y 54.7476, Z -8.0000, A 0.000, B 0.000, C 0.000 }
gfCNCPoint6[8337] = {X 369.7143, Y 54.2520, Z -8.0000, A 0.000, B 0.000, C 0.000 }
gfCNCPoint6[8338] = {X 370.5936, Y 53.9443, Z -8.0000, A 0.000, B 0.000, C 0.000 }
gfCNCPoint6[8339] = {X 371.5193, Y 53.8400, Z -8.0000, A 0.000, B 0.000, C 0.000 }
gfCNCPoint6[8340] = {X 388.0597, Y 53.8400, Z -8.0000, A 0.000, B 0.000, C 0.000 }
gfCNCPoint6[8341] = {X 388.9854, Y 53.9443, Z -8.0000, A 0.000, B 0.000, C 0.000 }
gfCNCPoint6[8342] = {X 389.8646, Y 54.2520, Z -8.0000, A 0.000, B 0.000, C 0.000 }
gfCNCPoint6[8343] = {X 390.6534, Y 54.7476, Z -8.0000, A 0.000, B 0.000, C 0.000 }
gfCNCPoint6[8344] = {X 391.3121, Y 55.4063, Z -8.0000, A 0.000, B 0.000, C 0.000 }
gfCNCPoint6[8345] = {X 391.8077, Y 56.1950, Z -8.0000, A 0.000, B 0.000, C 0.000 }
gfCNCPoint6[8346] = {X 392.1154, Y 57.0743, Z -8.0000, A 0.000, B 0.000, C 0.000 }
gfCNCPoint6[8347] = {X 392.2197, Y 58.0000, Z -8.0000, A 0.000, B 0.000, C 0.000 }
gfCNCPoint6[8348] = {X 392.2197, Y 58.9342, Z -8.0000, A 0.000, B 0.000, C 0.000 }
gfCNCPoint6[8349] = {X 392.1167, Y 59.8538, Z -8.0000, A 0.000, B 0.000, C 0.000 }
gfCNCPoint6[8350] = {X 391.8131, Y 60.7279, Z -8.0000, A 0.000, B 0.000, C 0.000 }
gfCNCPoint6[8351] = {X 391.3966, Y 61.4188, Z -8.0000, A 0.000, B 0.000, C 0.000 }
gfCNCPoint6[8352] = {X 390.8554, Y 62.0170, Z -8.0000, A 0.000, B 0.000, C 0.000 }
gfCNCPoint6[8353] = {X 390.2094, Y 62.5001, Z -8.0000, A 0.000, B 0.000, C 0.000 }
gfCNCPoint6[8354] = {X 389.4826, Y 62.8503, Z -8.0000, A 0.000, B 0.000, C 0.000 }
gfCNCPoint6[8355] = {X 388.7022, Y 63.0545, Z -8.0000, A 0.000, B 0.000, C 0.000 }
gfCNCPoint6[8356] = {X 388.6020, Y 63.0694, Z -8.0000, A 0.000, B 0.000, C 0.000 }
gfCNCPoint6[8357] = {X 388.5014, Y 63.0818, Z -8.0000, A 0.000, B 0.000, C 0.000 }
gfCNCPoint6[8358] = {X 388.4983, Y 84.6154, Z -8.0000, A 0.000, B 0.000, C 0.000 }
gfCNCPoint6[8359] = {X 388.4389, Y 86.2600, Z -8.0000, A 0.000, B 0.000, C 0.000 }
gfCNCPoint6[8360] = {X 388.2363, Y 87.8931, Z -8.0000, A 0.000, B 0.000, C 0.000 }
gfCNCPoint6[8361] = {X 387.8920, Y 89.5023, Z -8.0000, A 0.000, B 0.000, C 0.000 }
gfCNCPoint6[8362] = {X 387.3700, Y 91.0599, Z -8.0000, A 0.000, B 0.000, C 0.000 }
gfCNCPoint6[8363] = {X 386.6360, Y 92.5296, Z -8.0000, A 0.000, B 0.000, C 0.000 }
gfCNCPoint6[8364] = {X 385.7043, Y 93.8825, Z -8.0000, A 0.000, B 0.000, C 0.000 }
gfCNCPoint6[8365] = {X 384.5930, Y 95.0924, Z -8.0000, A 0.000, B 0.000, C 0.000 }
gfCNCPoint6[8366] = {X 383.0850, Y 96.3690, Z -8.0000, A 0.000, B 0.000, C 0.000 }
gfCNCPoint6[8367] = {X 381.4486, Y 97.4764, Z -8.0000, A 0.000, B 0.000, C 0.000 }
gfCNCPoint6[8368] = {X 379.7029, Y 98.4018, Z -8.0000, A 0.000, B 0.000, C 0.000 }
gfCNCPoint6[8369] = {X 377.4420, Y 99.3523, Z -8.0000, A 0.000, B 0.000, C 0.000 }
gfCNCPoint6[8370] = {X 375.1189, Y 100.1388, Z -8.0000, A 0.000, B 0.000, C 0.000 }
gfCNCPoint6[8371] = {X 372.7456, Y 100.7574, Z -8.0000, A 0.000, B 0.000, C 0.000 }
gfCNCPoint6[8372] = {X 369.0716, Y 101.4723, Z -8.0000, A 0.000, B 0.000, C 0.000 }
gfCNCPoint6[8373] = {X 365.3680, Y 102.0134, Z -8.0000, A 0.000, B 0.000, C 0.000 }
gfCNCPoint6[8374] = {X 361.6430, Y 102.3793, Z -8.0000, A 0.000, B 0.000, C 0.000 }
gfCNCPoint6[8375] = {X 355.6386, Y 102.7230, Z -8.0000, A 0.000, B 0.000, C 0.000 }
gfCNCPoint6[8376] = {X 349.6261, Y 102.8679, Z -8.0000, A 0.000, B 0.000, C 0.000 }
gfCNCPoint6[8377] = {X 349.6563, Y 106.8678, Z -8.0000, A 0.000, B 0.000, C 0.000 }
gfCNCPoint6[8378] = {X 349.6255, Y 102.7879, Z -8.0000, A 0.000, B 0.000, C 0.000 }
gfCNCPoint6[8379] = {X 345.9322, Y 102.7783, Z -8.0000, A 0.000, B 0.000, C 0.000 }
gfCNCPoint6[8380] = {X 342.2399, Y 102.6936, Z -8.0000, A 0.000, B 0.000, C 0.000 }
gfCNCPoint6[8381] = {X 337.6059, Y 102.5039, Z -8.0000, A 0.000, B 0.000, C 0.000 }
gfCNCPoint6[8382] = {X 332.9835, Y 102.1247, Z -8.0000, A 0.000, B 0.000, C 0.000 }
gfCNCPoint6[8383] = {X 328.3805, Y 101.5566, Z -8.0000, A 0.000, B 0.000, C 0.000 }
gfCNCPoint6[8384] = {X 325.3272, Y 101.0208, Z -8.0000, A 0.000, B 0.000, C 0.000 }
gfCNCPoint6[8385] = {X 322.3168, Y 100.2811, Z -8.0000, A 0.000, B 0.000, C 0.000 }
gfCNCPoint6[8386] = {X 319.3629, Y 99.3408, Z -8.0000, A 0.000, B 0.000, C 0.000 }
gfCNCPoint6[8387] = {X 317.6427, Y 98.6527, Z -8.0000, A 0.000, B 0.000, C 0.000 }
gfCNCPoint6[8388] = {X 315.9868, Y 97.8217, Z -8.0000, A 0.000, B 0.000, C 0.000 }
gfCNCPoint6[8389] = {X 314.4072, Y 96.8536, Z -8.0000, A 0.000, B 0.000, C 0.000 }
gfCNCPoint6[8390] = {X 312.9151, Y 95.7553, Z -8.0000, A 0.000, B 0.000, C 0.000 }
gfCNCPoint6[8391] = {X 311.7820, Y 94.7196, Z -8.0000, A 0.000, B 0.000, C 0.000 }
gfCNCPoint6[8392] = {X 310.7900, Y 93.5481, Z -8.0000, A 0.000, B 0.000, C 0.000 }
gfCNCPoint6[8393] = {X 309.9553, Y 92.2598, Z -8.0000, A 0.000, B 0.000, C 0.000 }
gfCNCPoint6[8394] = {X 309.2914, Y 90.8756, Z -8.0000, A 0.000, B 0.000, C 0.000 }
gfCNCPoint6[8395] = {X 308.7336, Y 89.0638, Z -8.0000, A 0.000, B 0.000, C 0.000 }
gfCNCPoint6[8396] = {X 308.3842, Y 87.2005, Z -8.0000, A 0.000, B 0.000, C 0.000 }
gfCNCPoint6[8397] = {X 308.2476, Y 85.3097, Z -8.0000, A 0.000, B 0.000, C 0.000 }
gfCNCPoint6[8398] = {X 308.2340, Y 84.6167, Z -8.0000, A 0.000, B 0.000, C 0.000 }
gfCNCPoint6[8399] = {X 308.2353, Y 62.9981, Z -8.0000, A 0.000, B 0.000, C 0.000 }
gfCNCPoint6[8400] = {X 307.3938, Y 62.8329, Z -8.0000, A 0.000, B 0.000, C 0.000 }
gfCNCPoint6[8401] = {X 306.6055, Y 62.4954, Z -8.0000, A 0.000, B 0.000, C 0.000 }
gfCNCPoint6[8402] = {X 305.9051, Y 62.0007, Z -8.0000, A 0.000, B 0.000, C 0.000 }
gfCNCPoint6[8403] = {X 305.3236, Y 61.3705, Z -8.0000, A 0.000, B 0.000, C 0.000 }
gfCNCPoint6[8404] = {X 304.8866, Y 60.6326, Z -8.0000, A 0.000, B 0.000, C 0.000 }
gfCNCPoint6[8405] = {X 304.6135, Y 59.8198, Z -8.0000, A 0.000, B 0.000, C 0.000 }
gfCNCPoint6[8406] = {X 304.5164, Y 58.9678, Z -8.0000, A 0.000, B 0.000, C 0.000 }
gfCNCPoint6[8407] = {X 304.5162, Y 58.0000, Z -8.0000, A 0.000, B 0.000, C 0.000 }
gfCNCPoint6[8408] = {X 304.6185, Y 57.0921, Z -8.0000, A 0.000, B 0.000, C 0.000 }
gfCNCPoint6[8409] = {X 304.9203, Y 56.2298, Z -8.0000, A 0.000, B 0.000, C 0.000 }
gfCNCPoint6[8410] = {X 305.4064, Y 55.4562, Z -8.0000, A 0.000, B 0.000, C 0.000 }
gfCNCPoint6[8411] = {X 306.0524, Y 54.8101, Z -8.0000, A 0.000, B 0.000, C 0.000 }
gfCNCPoint6[8412] = {X 306.8260, Y 54.3240, Z -8.0000, A 0.000, B 0.000, C 0.000 }
gfCNCPoint6[8413] = {X 307.6883, Y 54.0223, Z -8.0000, A 0.000, B 0.000, C 0.000 }
gfCNCPoint6[8414] = {X 308.5962, Y 53.9200, Z -8.0000, A 0.000, B 0.000, C 0.000 }
gfCNCPoint6[8415] = {X 324.3107, Y 53.9200, Z -8.0000, A 0.000, B 0.000, C 0.000 }
gfCNCPoint6[8416] = {X 325.2186, Y 54.0223, Z -8.0000, A 0.000, B 0.000, C 0.000 }
gfCNCPoint6[8417] = {X 326.0809, Y 54.3240, Z -8.0000, A 0.000, B 0.000, C 0.000 }
gfCNCPoint6[8418] = {X 326.8545, Y 54.8101, Z -8.0000, A 0.000, B 0.000, C 0.000 }
gfCNCPoint6[8419] = {X 327.5006, Y 55.4562, Z -8.0000, A 0.000, B 0.000, C 0.000 }
gfCNCPoint6[8420] = {X 327.9866, Y 56.2298, Z -8.0000, A 0.000, B 0.000, C 0.000 }
gfCNCPoint6[8421] = {X 328.2884, Y 57.0921, Z -8.0000, A 0.000, B 0.000, C 0.000 }
gfCNCPoint6[8422] = {X 328.3907, Y 58.0000, Z -8.0000, A 0.000, B 0.000, C 0.000 }
gfCNCPoint6[8423] = {X 328.3907, Y 58.9345, Z -8.0000, A 0.000, B 0.000, C 0.000 }
gfCNCPoint6[8424] = {X 328.2960, Y 59.7915, Z -8.0000, A 0.000, B 0.000, C 0.000 }
gfCNCPoint6[8425] = {X 328.0249, Y 60.6099, Z -8.0000, A 0.000, B 0.000, C 0.000 }
gfCNCPoint6[8426] = {X 327.5893, Y 61.3540, Z -8.0000, A 0.000, B 0.000, C 0.000 }
gfCNCPoint6[8427] = {X 327.0083, Y 61.9910, Z -8.0000, A 0.000, B 0.000, C 0.000 }
gfCNCPoint6[8428] = {X 326.3074, Y 62.4930, Z -8.0000, A 0.000, B 0.000, C 0.000 }
gfCNCPoint6[8429] = {X 325.5172, Y 62.8380, Z -8.0000, A 0.000, B 0.000, C 0.000 }
gfCNCPoint6[8430] = {X 324.6726, Y 63.0109, Z -8.0000, A 0.000, B 0.000, C 0.000 }
gfCNCPoint6[8431] = {X 324.6746, Y 83.2309, Z -8.0000, A 0.000, B 0.000, C 0.000 }
gfCNCPoint6[8432] = {X 324.6881, Y 84.6155, Z -8.0000, A 0.000, B 0.000, C 0.000 }
gfCNCPoint6[8433] = {X 324.7699, Y 85.8991, Z -8.0000, A 0.000, B 0.000, C 0.000 }
gfCNCPoint6[8434] = {X 325.0029, Y 87.1640, Z -8.0000, A 0.000, B 0.000, C 0.000 }
gfCNCPoint6[8435] = {X 325.5050, Y 87.6524, Z -8.0000, A 0.000, B 0.000, C 0.000 }
gfCNCPoint6[8436] = {X 326.1104, Y 88.0045, Z -8.0000, A 0.000, B 0.000, C 0.000 }
gfCNCPoint6[8437] = {X 327.9149, Y 88.7253, Z -8.0000, A 0.000, B 0.000, C 0.000 }
gfCNCPoint6[8438] = {X 329.7927, Y 89.2249, Z -8.0000, A 0.000, B 0.000, C 0.000 }
gfCNCPoint6[8439] = {X 332.8903, Y 89.7806, Z -8.0000, A 0.000, B 0.000, C 0.000 }
gfCNCPoint6[8440] = {X 336.0160, Y 90.1465, Z -8.0000, A 0.000, B 0.000, C 0.000 }
gfCNCPoint6[8441] = {X 340.3936, Y 90.4413, Z -8.0000, A 0.000, B 0.000, C 0.000 }
gfCNCPoint6[8442] = {X 344.7784, Y 90.5954, Z -8.0000, A 0.000, B 0.000, C 0.000 }
gfCNCPoint6[8443] = {X 349.1659, Y 90.6086, Z -8.0000, A 0.000, B 0.000, C 0.000 }
gfCNCPoint6[8444] = {X 353.3251, Y 90.5401, Z -8.0000, A 0.000, B 0.000, C 0.000 }
gfCNCPoint6[8445] = {X 357.4791, Y 90.3207, Z -8.0000, A 0.000, B 0.000, C 0.000 }
gfCNCPoint6[8446] = {X 361.6224, Y 89.9506, Z -8.0000, A 0.000, B 0.000, C 0.000 }
gfCNCPoint6[8447] = {X 363.7169, Y 89.6617, Z -8.0000, A 0.000, B 0.000, C 0.000 }
gfCNCPoint6[8448] = {X 365.7921, Y 89.2572, Z -8.0000, A 0.000, B 0.000, C 0.000 }
gfCNCPoint6[8449] = {X 367.8417, Y 88.7382, Z -8.0000, A 0.000, B 0.000, C 0.000 }
gfCNCPoint6[8450] = {X 368.7990, Y 88.4167, Z -8.0000, A 0.000, B 0.000, C 0.000 }
gfCNCPoint6[8451] = {X 369.7141, Y 87.9895, Z -8.0000, A 0.000, B 0.000, C 0.000 }
gfCNCPoint6[8452] = {X 370.5753, Y 87.4621, Z -8.0000, A 0.000, B 0.000, C 0.000 }
gfCNCPoint6[8453] = {X 370.7898, Y 87.2386, Z -8.0000, A 0.000, B 0.000, C 0.000 }
gfCNCPoint6[8454] = {X 370.9004, Y 86.9492, Z -8.0000, A 0.000, B 0.000, C 0.000 }
gfCNCPoint6[8455] = {X 371.0941, Y 85.3945, Z -8.0000, A 0.000, B 0.000, C 0.000 }
gfCNCPoint6[8456] = {X 371.1587, Y 83.8290, Z -8.0000, A 0.000, B 0.000, C 0.000 }
gfCNCPoint6[8457] = {X 371.1598, Y 62.9982, Z -8.0000, A 0.000, B 0.000, C 0.000 }
gfCNCPoint6[8458] = {X 371.0232, Y 62.9838, Z -8.0000, A 0.000, B 0.000, C 0.000 }
gfCNCPoint6[8459] = {X 370.8872, Y 62.9648, Z -8.0000, A 0.000, B 0.000, C 0.000 }
gfCNCPoint6[8460] = {X 369.9679, Y 62.7076, Z -8.0000, A 0.000, B 0.000, C 0.000 }
gfCNCPoint6[8461] = {X 369.1336, Y 62.2439, Z -8.0000, A 0.000, B 0.000, C 0.000 }
gfCNCPoint6[8462] = {X 368.4298, Y 61.5990, Z -8.0000, A 0.000, B 0.000, C 0.000 }
gfCNCPoint6[8463] = {X 367.8952, Y 60.8082, Z -8.0000, A 0.000, B 0.000, C 0.000 }
gfCNCPoint6[8464] = {X 367.5589, Y 59.9148, Z -8.0000, A 0.000, B 0.000, C 0.000 }
gfCNCPoint6[8465] = {X 367.4394, Y 58.9678, Z -8.0000, A 0.000, B 0.000, C 0.000 }
gfCNCPoint6[8466] = {X 367.4393, Y 58.0000, Z -8.0000, A 0.000, B 0.000, C 0.000 }
gfCNCPoint6[8467] = {X 367.5416, Y 57.0921, Z -8.0000, A 0.000, B 0.000, C 0.000 }
gfCNCPoint6[8468] = {X 367.8433, Y 56.2298, Z -8.0000, A 0.000, B 0.000, C 0.000 }
gfCNCPoint6[8469] = {X 368.3294, Y 55.4562, Z -8.0000, A 0.000, B 0.000, C 0.000 }
gfCNCPoint6[8470] = {X 368.9754, Y 54.8101, Z -8.0000, A 0.000, B 0.000, C 0.000 }
gfCNCPoint6[8471] = {X 369.7490, Y 54.3240, Z -8.0000, A 0.000, B 0.000, C 0.000 }
gfCNCPoint6[8472] = {X 370.6114, Y 54.0223, Z -8.0000, A 0.000, B 0.000, C 0.000 }
gfCNCPoint6[8473] = {X 371.5193, Y 53.9200, Z -8.0000, A 0.000, B 0.000, C 0.000 }
gfCNCPoint6[8474] = {X 388.0597, Y 53.9200, Z -8.0000, A 0.000, B 0.000, C 0.000 }
gfCNCPoint6[8475] = {X 388.9676, Y 54.0223, Z -8.0000, A 0.000, B 0.000, C 0.000 }
